LIN {X 0,Y 446.701,Z 503.839,A -85,B 0,C 180,E1 -8817.295,E2 -8817.295} C_VEL
LIN {X 0,Y 446.785,Z 503.811,A -85,B 0,C 180,E1 -8820,E2 -8820} C_VEL
LIN {X 0,Y 446.702,Z 503.837,A -85,B 0,C 180,E1 -8822.706,E2 -8822.706} C_VEL
LIN {X 0,Y 446.643,Z 503.843,A -85,B 0,C 180,E1 -8826.324,E2 -8826.324} C_VEL
LIN {X 0,Y 446.53,Z 503.851,A -85,B 0,C 180,E1 -8829.056,E2 -8829.056} C_VEL
LIN {X 0,Y 446.513,Z 503.865,A -85,B 0,C 180,E1 -8832.73,E2 -8832.73} C_VEL
LIN {X 0,Y 446.488,Z 503.852,A -85,B 0,C 180,E1 -8836.228,E2 -8836.228} C_VEL
LIN {X 0,Y 446.462,Z 503.873,A -85,B 0,C 180,E1 -8839.304,E2 -8839.304} C_VEL
LIN {X 0,Y 446.41,Z 503.87,A -85,B 0,C 180,E1 -8842.2,E2 -8842.2} C_VEL
LIN {X 0,Y 446.452,Z 503.872,A -85,B 0,C 180,E1 -8845.153,E2 -8845.153} C_VEL
LIN {X 0,Y 446.478,Z 503.864,A -85,B 0,C 180,E1 -8848.18,E2 -8848.18} C_VEL
LIN {X 0,Y 446.428,Z 503.877,A -85,B 0,C 180,E1 -8851.3,E2 -8851.3} C_VEL
LIN {X 0,Y 446.426,Z 503.872,A -85,B 0,C 180,E1 -8854.524,E2 -8854.524} C_VEL
LIN {X 0,Y 446.427,Z 503.874,A -85,B 0,C 180,E1 -8858.083,E2 -8858.083} C_VEL
LIN {X 0,Y 446.424,Z 503.878,A -85,B 0,C 180,E1 -8860.919,E2 -8860.919} C_VEL
LIN {X 0,Y 446.421,Z 503.873,A -85,B 0,C 180,E1 -8863.844,E2 -8863.844} C_VEL
LIN {X 0,Y 446.422,Z 503.876,A -85,B 0,C 180,E1 -8866.401,E2 -8866.401} C_VEL
LIN {X 0,Y 446.447,Z 503.87,A -85,B 0,C 180,E1 -8869.804,E2 -8869.804} C_VEL
LIN {X 0,Y 446.409,Z 503.874,A -85,B 0,C 180,E1 -8872.122,E2 -8872.122} C_VEL
LIN {X 0,Y 446.429,Z 503.873,A -85,B 0,C 180,E1 -8875.478,E2 -8875.478} C_VEL
LIN {X 0,Y 446.417,Z 503.875,A -85,B 0,C 180,E1 -8878.701,E2 -8878.701} C_VEL
LIN {X 0,Y 446.486,Z 503.868,A -85,B 0,C 180,E1 -8881.822,E2 -8881.822} C_VEL
LIN {X 0,Y 446.529,Z 503.926,A -85,B 0,C 180,E1 -8882.431,E2 -8882.431} C_VEL
LIN {X 0,Y 448.673,Z 514.714,A -85,B 0,C 180,E1 -8884.485,E2 -8884.485} C_VEL
LIN {X 0,Y 448.915,Z 519.545,A -85,B 0,C 180,E1 -8885.368,E2 -8885.368} C_VEL
LIN {X 0,Y 448.25,Z 538.154,A -85,B 0,C 180,E1 -8888.622,E2 -8888.622} C_VEL
LIN {X 0,Y 447.958,Z 547.38,A -85,B 0,C 180,E1 -8890.172,E2 -8890.172} C_VEL
LIN {X 0,Y 451.104,Z 565.732,A -85,B 0,C 180,E1 -8890.623,E2 -8890.623} C_VEL
LIN {X 0,Y 450.374,Z 639.656,A -85,B 0,C 180,E1 -8891.807,E2 -8891.807} C_VEL
LIN {X 0,Y 449.624,Z 645.502,A -85,B 0,C 180,E1 -8891.871,E2 -8891.871} C_VEL
LIN {X 0,Y 446.643,Z 654.974,A -85,B 0,C 180,E1 -8891.928,E2 -8891.928} C_VEL
LIN {X 0,Y 443.724,Z 664.359,A -85,B 0,C 180,E1 -8892.063,E2 -8892.063} C_VEL
LIN {X 0,Y 443.009,Z 670.054,A -85,B 0,C 180,E1 -8892.237,E2 -8892.237} C_VEL
LIN {X 0,Y 442.573,Z 683.413,A -85,B 0,C 180,E1 -8892.857,E2 -8892.857} C_VEL
LIN {X 0,Y 441.986,Z 695.4,A -85,B 0,C 180,E1 -8893.606,E2 -8893.606} C_VEL
LIN {X 0,Y 441.337,Z 706.738,A -85,B 0,C 180,E1 -8894.53,E2 -8894.53} C_VEL
LIN {X 0,Y 440.642,Z 716.953,A -85,B 0,C 180,E1 -8895.57,E2 -8895.57} C_VEL
LIN {X 0,Y 440.123,Z 725.673,A -85,B 0,C 180,E1 -8896.66,E2 -8896.66} C_VEL
LIN {X 0,Y 439.657,Z 734.405,A -85,B 0,C 180,E1 -8898.006,E2 -8898.006} C_VEL
LIN {X 0,Y 439.126,Z 741.667,A -85,B 0,C 180,E1 -8899.394,E2 -8899.394} C_VEL
LIN {X 0,Y 438.802,Z 747.491,A -85,B 0,C 180,E1 -8900.784,E2 -8900.784} C_VEL
LIN {X 0,Y 438.596,Z 752.07,A -85,B 0,C 180,E1 -8902.172,E2 -8902.172} C_VEL
LIN {X 0,Y 438.466,Z 755.655,A -85,B 0,C 180,E1 -8903.608,E2 -8903.608} C_VEL
LIN {X 0,Y 438.396,Z 757.307,A -85,B 0,C 180,E1 -8904.481,E2 -8904.481} C_VEL
LIN {X 0,Y 438.271,Z 759.557,A -85,B 0,C 180,E1 -8906.322,E2 -8906.322} C_VEL
LIN {X 0,Y 438.355,Z 760.102,A -85,B 0,C 180,E1 -8907.243,E2 -8907.243} C_VEL
LIN {X 0,Y 438.296,Z 760.224,A -85,B 0,C 180,E1 -8908.162,E2 -8908.162} C_VEL
LIN {X 0,Y 438.256,Z 759.301,A -85,B 0,C 180,E1 -8910,E2 -8910} C_VEL
LIN {X 0,Y 438.264,Z 758.263,A -85,B 0,C 180,E1 -8910.919,E2 -8910.919} C_VEL
LIN {X 0,Y 438.373,Z 756.774,A -85,B 0,C 180,E1 -8911.837,E2 -8911.837} C_VEL
LIN {X 0,Y 438.55,Z 753.771,A -85,B 0,C 180,E1 -8913.215,E2 -8913.215} C_VEL
LIN {X 0,Y 438.677,Z 749.73,A -85,B 0,C 180,E1 -8914.594,E2 -8914.594} C_VEL
LIN {X 0,Y 438.925,Z 744.532,A -85,B 0,C 180,E1 -8915.974,E2 -8915.974} C_VEL
LIN {X 0,Y 439.352,Z 738.014,A -85,B 0,C 180,E1 -8917.352,E2 -8917.352} C_VEL
LIN {X 0,Y 439.795,Z 729.922,A -85,B 0,C 180,E1 -8918.732,E2 -8918.732} C_VEL
LIN {X 0,Y 440.32,Z 721.586,A -85,B 0,C 180,E1 -8919.88,E2 -8919.88} C_VEL
LIN {X 0,Y 441.004,Z 711.36,A -85,B 0,C 180,E1 -8921.025,E2 -8921.025} C_VEL
LIN {X 0,Y 441.496,Z 701.275,A -85,B 0,C 180,E1 -8921.943,E2 -8921.943} C_VEL
LIN {X 0,Y 442.074,Z 690.211,A -85,B 0,C 180,E1 -8922.743,E2 -8922.743} C_VEL
LIN {X 0,Y 442.675,Z 677.742,A -85,B 0,C 180,E1 -8923.426,E2 -8923.426} C_VEL
LIN {X 0,Y 443.015,Z 664.927,A -85,B 0,C 180,E1 -8923.935,E2 -8923.935} C_VEL
LIN {X 0,Y 443.262,Z 651.37,A -85,B 0,C 180,E1 -8924.265,E2 -8924.265} C_VEL
LIN {X 0,Y 444.008,Z 565.064,A -85,B 0,C 180,E1 -8925.668,E2 -8925.668} C_VEL
LIN {X 0,Y 440.929,Z 547.62,A -85,B 0,C 180,E1 -8926.085,E2 -8926.085} C_VEL
LIN {X 0,Y 441.452,Z 530.278,A -85,B 0,C 180,E1 -8929.048,E2 -8929.048} C_VEL
LIN {X 0,Y 441.954,Z 517.971,A -85,B 0,C 180,E1 -8931.209,E2 -8931.209} C_VEL
LIN {X 0,Y 439.439,Z 504.755,A -85,B 0,C 180,E1 -8933.719,E2 -8933.719} C_VEL
LIN {X 0,Y 439.431,Z 504.751,A -85,B 0,C 180,E1 -8936.603,E2 -8936.603} C_VEL
LIN {X 0,Y 439.384,Z 504.754,A -85,B 0,C 180,E1 -8939.725,E2 -8939.725} C_VEL
LIN {X 0,Y 439.374,Z 504.757,A -85,B 0,C 180,E1 -8942.945,E2 -8942.945} C_VEL
LIN {X 0,Y 439.373,Z 504.752,A -85,B 0,C 180,E1 -8946.286,E2 -8946.286} C_VEL
LIN {X 0,Y 439.4,Z 504.745,A -85,B 0,C 180,E1 -8949.848,E2 -8949.848} C_VEL
LIN {X 0,Y 439.398,Z 504.753,A -85,B 0,C 180,E1 -8952.628,E2 -8952.628} C_VEL
LIN {X 0,Y 439.405,Z 504.744,A -85,B 0,C 180,E1 -8955.271,E2 -8955.271} C_VEL
LIN {X 0,Y 439.386,Z 504.756,A -85,B 0,C 180,E1 -8958.742,E2 -8958.742} C_VEL
LIN {X 0,Y 439.381,Z 504.752,A -85,B 0,C 180,E1 -8961.605,E2 -8961.605} C_VEL
LIN {X 0,Y 439.396,Z 504.755,A -85,B 0,C 180,E1 -8964.843,E2 -8964.843} C_VEL
LIN {X 0,Y 439.455,Z 504.746,A -85,B 0,C 180,E1 -8966.016,E2 -8966.016} C_VEL
LIN {X 0,Y 443.719,Z 518.661,A -85,B 0,C 180,E1 -8966.455,E2 -8966.455} C_VEL
LIN {X 0,Y 444.068,Z 521.82,A -85,B 0,C 180,E1 -8966.527,E2 -8966.527} C_VEL
LIN {X 0,Y 442.839,Z 611.676,A -85,B 0,C 180,E1 -8968.15,E2 -8968.15} C_VEL
LIN {X 0,Y 442.549,Z 625.742,A -85,B 0,C 180,E1 -8968.604,E2 -8968.604} C_VEL
LIN {X 0,Y 442.193,Z 638.28,A -85,B 0,C 180,E1 -8969.204,E2 -8969.204} C_VEL
LIN {X 0,Y 441.679,Z 649.543,A -85,B 0,C 180,E1 -8969.918,E2 -8969.918} C_VEL
LIN {X 0,Y 441.128,Z 661.441,A -85,B 0,C 180,E1 -8970.883,E2 -8970.883} C_VEL
LIN {X 0,Y 440.621,Z 671.687,A -85,B 0,C 180,E1 -8971.931,E2 -8971.931} C_VEL
LIN {X 0,Y 440.071,Z 681.545,A -85,B 0,C 180,E1 -8973.182,E2 -8973.182} C_VEL
LIN {X 0,Y 439.609,Z 689.541,A -85,B 0,C 180,E1 -8974.427,E2 -8974.427} C_VEL
LIN {X 0,Y 439.275,Z 696.549,A -85,B 0,C 180,E1 -8975.773,E2 -8975.773} C_VEL
LIN {X 0,Y 439.002,Z 701.366,A -85,B 0,C 180,E1 -8976.907,E2 -8976.907} C_VEL
LIN {X 0,Y 438.794,Z 706.406,A -85,B 0,C 180,E1 -8978.384,E2 -8978.384} C_VEL
LIN {X 0,Y 438.609,Z 710.13,A -85,B 0,C 180,E1 -8979.848,E2 -8979.848} C_VEL
LIN {X 0,Y 438.443,Z 712.707,A -85,B 0,C 180,E1 -8981.301,E2 -8981.301} C_VEL
LIN {X 0,Y 438.377,Z 713.822,A -85,B 0,C 180,E1 -8982.265,E2 -8982.265} C_VEL
LIN {X 0,Y 438.384,Z 714.51,A -85,B 0,C 180,E1 -8983.227,E2 -8983.227} C_VEL
LIN {X 0,Y 438.393,Z 714.74,A -85,B 0,C 180,E1 -8984.185,E2 -8984.185} C_VEL
LIN {X 0,Y 438.388,Z 714.513,A -85,B 0,C 180,E1 -8985.137,E2 -8985.137} C_VEL
LIN {X 0,Y 438.443,Z 713.872,A -85,B 0,C 180,E1 -8986.087,E2 -8986.087} C_VEL
LIN {X 0,Y 438.606,Z 711.588,A -85,B 0,C 180,E1 -8987.798,E2 -8987.798} C_VEL
LIN {X 0,Y 438.817,Z 708.09,A -85,B 0,C 180,E1 -8989.386,E2 -8989.386} C_VEL
LIN {X 0,Y 439.028,Z 703.85,A -85,B 0,C 180,E1 -8990.788,E2 -8990.788} C_VEL
LIN {X 0,Y 439.373,Z 698.201,A -85,B 0,C 180,E1 -8992.232,E2 -8992.232} C_VEL
LIN {X 0,Y 439.806,Z 691.572,A -85,B 0,C 180,E1 -8993.577,E2 -8993.577} C_VEL
LIN {X 0,Y 440.275,Z 683.036,A -85,B 0,C 180,E1 -8994.963,E2 -8994.963} C_VEL
LIN {X 0,Y 440.812,Z 674.257,A -85,B 0,C 180,E1 -8996.114,E2 -8996.114} C_VEL
LIN {X 0,Y 441.367,Z 663.485,A -85,B 0,C 180,E1 -8997.262,E2 -8997.262} C_VEL
LIN {X 0,Y 441.962,Z 652.565,A -85,B 0,C 180,E1 -8998.177,E2 -8998.177} C_VEL
LIN {X 0,Y 442.557,Z 640.376,A -85,B 0,C 180,E1 -8998.976,E2 -8998.976} C_VEL
LIN {X 0,Y 442.923,Z 627.861,A -85,B 0,C 180,E1 -8999.592,E2 -8999.592} C_VEL
LIN {X 0,Y 443.21,Z 615.153,A -85,B 0,C 180,E1 -9000.022,E2 -9000.022} C_VEL
LIN {X 0,Y 443.443,Z 594.465,A -85,B 0,C 180,E1 -9000.437,E2 -9000.437} C_VEL
LIN {X 0,Y 444.597,Z 520.546,A -85,B 0,C 180,E1 -9001.826,E2 -9001.826} C_VEL
LIN {X 0,Y 443.026,Z 515.39,A -85,B 0,C 180,E1 -9002.01,E2 -9002.01} C_VEL
LIN {X 0,Y 440.276,Z 508.037,A -85,B 0,C 180,E1 -9002.302,E2 -9002.302} C_VEL
LIN {X 0,Y 439.499,Z 504.741,A -85,B 0,C 180,E1 -9003.323,E2 -9003.323} C_VEL
LIN {X 0,Y 439.614,Z 504.725,A -85,B 0,C 180,E1 -9006.425,E2 -9006.425} C_VEL
LIN {X 0,Y 439.493,Z 504.743,A -85,B 0,C 180,E1 -9009.202,E2 -9009.202} C_VEL
LIN {X 0,Y 439.495,Z 504.739,A -85,B 0,C 180,E1 -9012.727,E2 -9012.727} C_VEL
LIN {X 0,Y 439.438,Z 504.745,A -85,B 0,C 180,E1 -9016.349,E2 -9016.349} C_VEL
LIN {X 0,Y 439.394,Z 504.751,A -85,B 0,C 180,E1 -9019.627,E2 -9019.627} C_VEL
LIN {X 0,Y 439.357,Z 504.756,A -85,B 0,C 180,E1 -9022.576,E2 -9022.576} C_VEL
LIN {X 0,Y 439.397,Z 504.749,A -85,B 0,C 180,E1 -9025.585,E2 -9025.585} C_VEL
LIN {X 0,Y 439.418,Z 504.746,A -85,B 0,C 180,E1 -9028.673,E2 -9028.673} C_VEL
LIN {X 0,Y 439.367,Z 504.75,A -85,B 0,C 180,E1 -9031.861,E2 -9031.861} C_VEL
LIN {X 0,Y 439.394,Z 504.753,A -85,B 0,C 180,E1 -9035.156,E2 -9035.156} C_VEL
LIN {X 0,Y 439.384,Z 504.751,A -85,B 0,C 180,E1 -9038.595,E2 -9038.595} C_VEL
LIN {X 0,Y 439.383,Z 504.755,A -85,B 0,C 180,E1 -9041.257,E2 -9041.257} C_VEL
LIN {X 0,Y 439.397,Z 504.753,A -85,B 0,C 180,E1 -9044.73,E2 -9044.73} C_VEL
LIN {X 0,Y 439.394,Z 504.752,A -85,B 0,C 180,E1 -9047.797,E2 -9047.797} C_VEL
LIN {X 0,Y 439.427,Z 504.749,A -85,B 0,C 180,E1 -9050.229,E2 -9050.229} C_VEL
LIN {X 0,Y 439.374,Z 504.754,A -85,B 0,C 180,E1 -9053.714,E2 -9053.714} C_VEL
LIN {X 0,Y 439.371,Z 504.761,A -85,B 0,C 180,E1 -9057.055,E2 -9057.055} C_VEL
LIN {X 0,Y 439.434,Z 504.811,A -85,B 0,C 180,E1 -9060.887,E2 -9060.887} C_VEL
LIN {X 0,Y 441.948,Z 516.24,A -85,B 0,C 180,E1 -9063.169,E2 -9063.169} C_VEL
LIN {X 0,Y 442.844,Z 522.646,A -85,B 0,C 180,E1 -9064.377,E2 -9064.377} C_VEL
LIN {X 0,Y 441.66,Z 542.589,A -85,B 0,C 180,E1 -9067.795,E2 -9067.795} C_VEL
LIN {X 0,Y 440.607,Z 562.702,A -85,B 0,C 180,E1 -9071.156,E2 -9071.156} C_VEL
LIN {X 0,Y 440.45,Z 566.137,A -85,B 0,C 180,E1 -9071.705,E2 -9071.705} C_VEL
LIN {X 0,Y 443.689,Z 590.86,A -85,B 0,C 180,E1 -9072.348,E2 -9072.348} C_VEL
LIN {X 0,Y 443.939,Z 596.387,A -85,B 0,C 180,E1 -9072.466,E2 -9072.466} C_VEL
LIN {X 0,Y 442.814,Z 677.088,A -85,B 0,C 180,E1 -9073.963,E2 -9073.963} C_VEL
LIN {X 0,Y 442.19,Z 695.595,A -85,B 0,C 180,E1 -9074.561,E2 -9074.561} C_VEL
LIN {X 0,Y 441.694,Z 707.963,A -85,B 0,C 180,E1 -9075.134,E2 -9075.134} C_VEL
LIN {X 0,Y 441.141,Z 718.982,A -85,B 0,C 180,E1 -9075.822,E2 -9075.822} C_VEL
LIN {X 0,Y 440.644,Z 730.447,A -85,B 0,C 180,E1 -9076.745,E2 -9076.745} C_VEL
LIN {X 0,Y 440.053,Z 740.763,A -85,B 0,C 180,E1 -9077.783,E2 -9077.783} C_VEL
LIN {X 0,Y 439.487,Z 749.99,A -85,B 0,C 180,E1 -9078.937,E2 -9078.937} C_VEL
LIN {X 0,Y 439.03,Z 758.938,A -85,B 0,C 180,E1 -9080.324,E2 -9080.324} C_VEL
LIN {X 0,Y 438.735,Z 766.108,A -85,B 0,C 180,E1 -9081.711,E2 -9081.711} C_VEL
LIN {X 0,Y 438.52,Z 771.792,A -85,B 0,C 180,E1 -9083.097,E2 -9083.097} C_VEL
LIN {X 0,Y 438.431,Z 776.248,A -85,B 0,C 180,E1 -9084.481,E2 -9084.481} C_VEL
LIN {X 0,Y 438.378,Z 778.591,A -85,B 0,C 180,E1 -9085.402,E2 -9085.402} C_VEL
LIN {X 0,Y 438.308,Z 780.499,A -85,B 0,C 180,E1 -9086.323,E2 -9086.323} C_VEL
LIN {X 0,Y 438.417,Z 781.956,A -85,B 0,C 180,E1 -9087.244,E2 -9087.244} C_VEL
LIN {X 0,Y 438.263,Z 783.597,A -85,B 0,C 180,E1 -9089.081,E2 -9089.081} C_VEL
LIN {X 0,Y 438.266,Z 783.831,A -85,B 0,C 180,E1 -9090,E2 -9090} C_VEL
LIN {X 0,Y 438.262,Z 783.624,A -85,B 0,C 180,E1 -9090.919,E2 -9090.919} C_VEL
LIN {X 0,Y 438.419,Z 782.018,A -85,B 0,C 180,E1 -9092.756,E2 -9092.756} C_VEL
LIN {X 0,Y 438.312,Z 780.602,A -85,B 0,C 180,E1 -9093.677,E2 -9093.677} C_VEL
LIN {X 0,Y 438.432,Z 777.642,A -85,B 0,C 180,E1 -9095.058,E2 -9095.058} C_VEL
LIN {X 0,Y 438.471,Z 773.619,A -85,B 0,C 180,E1 -9096.442,E2 -9096.442} C_VEL
LIN {X 0,Y 438.686,Z 767.398,A -85,B 0,C 180,E1 -9098.058,E2 -9098.058} C_VEL
LIN {X 0,Y 439.013,Z 760.611,A -85,B 0,C 180,E1 -9099.444,E2 -9099.444} C_VEL
LIN {X 0,Y 439.431,Z 752.134,A -85,B 0,C 180,E1 -9100.831,E2 -9100.831} C_VEL
LIN {X 0,Y 439.956,Z 743.389,A -85,B 0,C 180,E1 -9101.985,E2 -9101.985} C_VEL
LIN {X 0,Y 440.532,Z 733.532,A -85,B 0,C 180,E1 -9103.047,E2 -9103.047} C_VEL
LIN {X 0,Y 441.063,Z 723.244,A -85,B 0,C 180,E1 -9103.946,E2 -9103.946} C_VEL
LIN {X 0,Y 441.657,Z 711.46,A -85,B 0,C 180,E1 -9104.75,E2 -9104.75} C_VEL
LIN {X 0,Y 442.178,Z 699.172,A -85,B 0,C 180,E1 -9105.38,E2 -9105.38} C_VEL
LIN {X 0,Y 442.641,Z 686.478,A -85,B 0,C 180,E1 -9105.836,E2 -9105.836} C_VEL
LIN {X 0,Y 442.895,Z 672.991,A -85,B 0,C 180,E1 -9106.122,E2 -9106.122} C_VEL
LIN {X 0,Y 443.536,Z 608.774,A -85,B 0,C 180,E1 -9107.2,E2 -9107.2} C_VEL
LIN {X 0,Y 443.59,Z 591.986,A -85,B 0,C 180,E1 -9107.509,E2 -9107.509} C_VEL
LIN {X 0,Y 440.47,Z 568.609,A -85,B 0,C 180,E1 -9108.079,E2 -9108.079} C_VEL
LIN {X 0,Y 441.403,Z 549.446,A -85,B 0,C 180,E1 -9111.236,E2 -9111.236} C_VEL
LIN {X 0,Y 442.511,Z 530.547,A -85,B 0,C 180,E1 -9114.389,E2 -9114.389} C_VEL
LIN {X 0,Y 442.898,Z 521.782,A -85,B 0,C 180,E1 -9115.872,E2 -9115.872} C_VEL
LIN {X 0,Y 440.519,Z 509.778,A -85,B 0,C 180,E1 -9118.075,E2 -9118.075} C_VEL
LIN {X 0,Y 439.443,Z 504.749,A -85,B 0,C 180,E1 -9119.063,E2 -9119.063} C_VEL
LIN {X 0,Y 439.371,Z 504.758,A -85,B 0,C 180,E1 -9122.945,E2 -9122.945} C_VEL
LIN {X 0,Y 439.371,Z 504.749,A -85,B 0,C 180,E1 -9126.286,E2 -9126.286} C_VEL
LIN {X 0,Y 439.41,Z 504.745,A -85,B 0,C 180,E1 -9129.85,E2 -9129.85} C_VEL
LIN {X 0,Y 439.383,Z 504.753,A -85,B 0,C 180,E1 -9132.627,E2 -9132.627} C_VEL
LIN {X 0,Y 439.398,Z 504.755,A -85,B 0,C 180,E1 -9135.27,E2 -9135.27} C_VEL
LIN {X 0,Y 439.393,Z 504.745,A -85,B 0,C 180,E1 -9138.741,E2 -9138.741} C_VEL
LIN {X 0,Y 439.385,Z 504.75,A -85,B 0,C 180,E1 -9141.604,E2 -9141.604} C_VEL
LIN {X 0,Y 439.394,Z 504.747,A -85,B 0,C 180,E1 -9144.844,E2 -9144.844} C_VEL
LIN {X 0,Y 439.367,Z 504.747,A -85,B 0,C 180,E1 -9148.139,E2 -9148.139} C_VEL
LIN {X 0,Y 439.418,Z 504.751,A -85,B 0,C 180,E1 -9151.327,E2 -9151.327} C_VEL
LIN {X 0,Y 439.397,Z 504.745,A -85,B 0,C 180,E1 -9154.415,E2 -9154.415} C_VEL
LIN {X 0,Y 439.356,Z 504.753,A -85,B 0,C 180,E1 -9157.424,E2 -9157.424} C_VEL
LIN {X 0,Y 439.433,Z 504.745,A -85,B 0,C 180,E1 -9160.662,E2 -9160.662} C_VEL
LIN {X 0,Y 439.453,Z 504.73,A -85,B 0,C 180,E1 -9164.224,E2 -9164.224} C_VEL
LIN {X 0,Y 439.499,Z 504.735,A -85,B 0,C 180,E1 -9168.002,E2 -9168.002} C_VEL
LIN {X 0,Y 439.539,Z 504.718,A -85,B 0,C 180,E1 -9171.726,E2 -9171.726} C_VEL
LIN {X 0,Y 439.619,Z 504.719,A -85,B 0,C 180,E1 -9174.496,E2 -9174.496} C_VEL
LIN {X 0,Y 439.627,Z 504.715,A -85,B 0,C 180,E1 -9178.168,E2 -9178.168} C_VEL
LIN {X 0,Y 439.755,Z 504.686,A -85,B 0,C 180,E1 -9180,E2 -9180} C_VEL
LIN {X 0,Y 439.649,Z 504.716,A -85,B 0,C 180,E1 -9182.749,E2 -9182.749} C_VEL
LIN {X 0,Y 439.614,Z 504.719,A -85,B 0,C 180,E1 -9186.426,E2 -9186.426} C_VEL
LIN {X 0,Y 439.492,Z 504.729,A -85,B 0,C 180,E1 -9189.202,E2 -9189.202} C_VEL
LIN {X 0,Y 439.457,Z 504.747,A -85,B 0,C 180,E1 -9192.938,E2 -9192.938} C_VEL
LIN {X 0,Y 439.439,Z 504.73,A -85,B 0,C 180,E1 -9196.349,E2 -9196.349} C_VEL
LIN {X 0,Y 439.395,Z 504.75,A -85,B 0,C 180,E1 -9199.627,E2 -9199.627} C_VEL
LIN {X 0,Y 439.357,Z 504.751,A -85,B 0,C 180,E1 -9202.576,E2 -9202.576} C_VEL
LIN {X 0,Y 439.399,Z 504.75,A -85,B 0,C 180,E1 -9205.586,E2 -9205.586} C_VEL
LIN {X 0,Y 439.419,Z 504.746,A -85,B 0,C 180,E1 -9208.674,E2 -9208.674} C_VEL
LIN {X 0,Y 439.379,Z 504.751,A -85,B 0,C 180,E1 -9212.034,E2 -9212.034} C_VEL
LIN {X 0,Y 439.392,Z 504.75,A -85,B 0,C 180,E1 -9215.342,E2 -9215.342} C_VEL
LIN {X 0,Y 439.385,Z 504.754,A -85,B 0,C 180,E1 -9218.595,E2 -9218.595} C_VEL
LIN {X 0,Y 439.385,Z 504.758,A -85,B 0,C 180,E1 -9221.258,E2 -9221.258} C_VEL
LIN {X 0,Y 439.404,Z 504.751,A -85,B 0,C 180,E1 -9224.729,E2 -9224.729} C_VEL
LIN {X 0,Y 439.397,Z 504.749,A -85,B 0,C 180,E1 -9227.797,E2 -9227.797} C_VEL
LIN {X 0,Y 439.429,Z 504.744,A -85,B 0,C 180,E1 -9230.229,E2 -9230.229} C_VEL
LIN {X 0,Y 439.373,Z 504.752,A -85,B 0,C 180,E1 -9233.714,E2 -9233.714} C_VEL
LIN {X 0,Y 439.373,Z 504.755,A -85,B 0,C 180,E1 -9237.055,E2 -9237.055} C_VEL
LIN {X 0,Y 439.384,Z 504.752,A -85,B 0,C 180,E1 -9240.275,E2 -9240.275} C_VEL
LIN {X 0,Y 439.482,Z 504.873,A -85,B 0,C 180,E1 -9242.194,E2 -9242.194} C_VEL
LIN {X 0,Y 441.934,Z 517.239,A -85,B 0,C 180,E1 -9244.573,E2 -9244.573} C_VEL
LIN {X 0,Y 441.822,Z 525.514,A -85,B 0,C 180,E1 -9246.07,E2 -9246.07} C_VEL
LIN {X 0,Y 441.178,Z 542.313,A -85,B 0,C 180,E1 -9248.997,E2 -9248.997} C_VEL
LIN {X 0,Y 441.052,Z 547.544,A -85,B 0,C 180,E1 -9249.879,E2 -9249.879} C_VEL
LIN {X 0,Y 444.354,Z 565.884,A -85,B 0,C 180,E1 -9250.34,E2 -9250.34} C_VEL
LIN {X 0,Y 443.385,Z 656.466,A -85,B 0,C 180,E1 -9251.834,E2 -9251.834} C_VEL
LIN {X 0,Y 443.021,Z 669.411,A -85,B 0,C 180,E1 -9252.214,E2 -9252.214} C_VEL
LIN {X 0,Y 443.009,Z 670.054,A -85,B 0,C 180,E1 -9252.237,E2 -9252.237} C_VEL
LIN {X 0,Y 442.219,Z 675.707,A -85,B 0,C 180,E1 -9252.44,E2 -9252.44} C_VEL
LIN {X 0,Y 439.059,Z 684.741,A -85,B 0,C 180,E1 -9252.79,E2 -9252.79} C_VEL
LIN {X 0,Y 435.844,Z 693.491,A -85,B 0,C 180,E1 -9253.239,E2 -9253.239} C_VEL
LIN {X 0,Y 434.972,Z 698.627,A -85,B 0,C 180,E1 -9253.597,E2 -9253.597} C_VEL
LIN {X 0,Y 434.304,Z 709.182,A -85,B 0,C 180,E1 -9254.514,E2 -9254.514} C_VEL
LIN {X 0,Y 433.676,Z 717.981,A -85,B 0,C 180,E1 -9255.453,E2 -9255.453} C_VEL
LIN {X 0,Y 433.108,Z 727.033,A -85,B 0,C 180,E1 -9256.631,E2 -9256.631} C_VEL
LIN {X 0,Y 432.578,Z 735.79,A -85,B 0,C 180,E1 -9258.045,E2 -9258.045} C_VEL
LIN {X 0,Y 432.029,Z 742.845,A -85,B 0,C 180,E1 -9259.455,E2 -9259.455} C_VEL
LIN {X 0,Y 431.749,Z 747.598,A -85,B 0,C 180,E1 -9260.632,E2 -9260.632} C_VEL
LIN {X 0,Y 431.525,Z 752.195,A -85,B 0,C 180,E1 -9262.043,E2 -9262.043} C_VEL
LIN {X 0,Y 431.373,Z 756.075,A -85,B 0,C 180,E1 -9263.633,E2 -9263.633} C_VEL
LIN {X 0,Y 431.234,Z 758.791,A -85,B 0,C 180,E1 -9265.326,E2 -9265.326} C_VEL
LIN {X 0,Y 431.263,Z 760.283,A -85,B 0,C 180,E1 -9267.198,E2 -9267.198} C_VEL
LIN {X 0,Y 431.22,Z 760.418,A -85,B 0,C 180,E1 -9268.132,E2 -9268.132} C_VEL
LIN {X 0,Y 431.17,Z 759.51,A -85,B 0,C 180,E1 -9270,E2 -9270} C_VEL
LIN {X 0,Y 431.182,Z 758.482,A -85,B 0,C 180,E1 -9270.934,E2 -9270.934} C_VEL
LIN {X 0,Y 431.294,Z 757.005,A -85,B 0,C 180,E1 -9271.868,E2 -9271.868} C_VEL
LIN {X 0,Y 431.483,Z 754.016,A -85,B 0,C 180,E1 -9273.268,E2 -9273.268} C_VEL
LIN {X 0,Y 431.598,Z 749.992,A -85,B 0,C 180,E1 -9274.67,E2 -9274.67} C_VEL
LIN {X 0,Y 431.884,Z 744.811,A -85,B 0,C 180,E1 -9276.072,E2 -9276.072} C_VEL
LIN {X 0,Y 432.32,Z 738.311,A -85,B 0,C 180,E1 -9277.472,E2 -9277.472} C_VEL
LIN {X 0,Y 432.794,Z 730.246,A -85,B 0,C 180,E1 -9278.874,E2 -9278.874} C_VEL
LIN {X 0,Y 433.351,Z 721.941,A -85,B 0,C 180,E1 -9280.04,E2 -9280.04} C_VEL
LIN {X 0,Y 434.053,Z 711.745,A -85,B 0,C 180,E1 -9281.203,E2 -9281.203} C_VEL
LIN {X 0,Y 434.565,Z 701.699,A -85,B 0,C 180,E1 -9282.136,E2 -9282.136} C_VEL
LIN {X 0,Y 435.186,Z 690.712,A -85,B 0,C 180,E1 -9282.948,E2 -9282.948} C_VEL
LIN {X 0,Y 435.798,Z 678.336,A -85,B 0,C 180,E1 -9283.642,E2 -9283.642} C_VEL
LIN {X 0,Y 436.183,Z 665.11,A -85,B 0,C 180,E1 -9284.177,E2 -9284.177} C_VEL
LIN {X 0,Y 436.411,Z 652.341,A -85,B 0,C 180,E1 -9284.498,E2 -9284.498} C_VEL
LIN {X 0,Y 437.299,Z 566.356,A -85,B 0,C 180,E1 -9285.915,E2 -9285.915} C_VEL
LIN {X 0,Y 434.044,Z 547.715,A -85,B 0,C 180,E1 -9286.37,E2 -9286.37} C_VEL
LIN {X 0,Y 434.548,Z 530.393,A -85,B 0,C 180,E1 -9289.362,E2 -9289.362} C_VEL
LIN {X 0,Y 435.03,Z 519.325,A -85,B 0,C 180,E1 -9291.314,E2 -9291.314} C_VEL
LIN {X 0,Y 432.4,Z 505.631,A -85,B 0,C 180,E1 -9293.974,E2 -9293.974} C_VEL
LIN {X 0,Y 432.393,Z 505.626,A -85,B 0,C 180,E1 -9297.071,E2 -9297.071} C_VEL
LIN {X 0,Y 432.349,Z 505.632,A -85,B 0,C 180,E1 -9300.51,E2 -9300.51} C_VEL
LIN {X 0,Y 432.36,Z 505.624,A -85,B 0,C 180,E1 -9304.003,E2 -9304.003} C_VEL
LIN {X 0,Y 432.322,Z 505.633,A -85,B 0,C 180,E1 -9307.196,E2 -9307.196} C_VEL
LIN {X 0,Y 432.332,Z 505.626,A -85,B 0,C 180,E1 -9310.178,E2 -9310.178} C_VEL
LIN {X 0,Y 432.362,Z 505.629,A -85,B 0,C 180,E1 -9313.054,E2 -9313.054} C_VEL
LIN {X 0,Y 432.34,Z 505.622,A -85,B 0,C 180,E1 -9315.662,E2 -9315.662} C_VEL
LIN {X 0,Y 432.331,Z 505.632,A -85,B 0,C 180,E1 -9318.397,E2 -9318.397} C_VEL
LIN {X 0,Y 432.343,Z 505.628,A -85,B 0,C 180,E1 -9321.85,E2 -9321.85} C_VEL
LIN {X 0,Y 432.352,Z 505.631,A -85,B 0,C 180,E1 -9325.324,E2 -9325.324} C_VEL
LIN {X 0,Y 432.38,Z 505.626,A -85,B 0,C 180,E1 -9325.747,E2 -9325.747} C_VEL
LIN {X 0,Y 436.927,Z 519.644,A -85,B 0,C 180,E1 -9326.21,E2 -9326.21} C_VEL
LIN {X 0,Y 437.213,Z 524.529,A -85,B 0,C 180,E1 -9326.314,E2 -9326.314} C_VEL
LIN {X 0,Y 435.961,Z 612.071,A -85,B 0,C 180,E1 -9327.928,E2 -9327.928} C_VEL
LIN {X 0,Y 435.658,Z 625.901,A -85,B 0,C 180,E1 -9328.38,E2 -9328.38} C_VEL
LIN {X 0,Y 435.28,Z 639.165,A -85,B 0,C 180,E1 -9329.025,E2 -9329.025} C_VEL
LIN {X 0,Y 434.729,Z 650.87,A -85,B 0,C 180,E1 -9329.789,E2 -9329.789} C_VEL
LIN {X 0,Y 434.207,Z 661.679,A -85,B 0,C 180,E1 -9330.684,E2 -9330.684} C_VEL
LIN {X 0,Y 433.683,Z 671.641,A -85,B 0,C 180,E1 -9331.705,E2 -9331.705} C_VEL
LIN {X 0,Y 433.114,Z 681.615,A -85,B 0,C 180,E1 -9332.977,E2 -9332.977} C_VEL
LIN {X 0,Y 432.638,Z 689.7,A -85,B 0,C 180,E1 -9334.244,E2 -9334.244} C_VEL
LIN {X 0,Y 432.281,Z 696.569,A -85,B 0,C 180,E1 -9335.564,E2 -9335.564} C_VEL
LIN {X 0,Y 431.928,Z 702.625,A -85,B 0,C 180,E1 -9337.013,E2 -9337.013} C_VEL
LIN {X 0,Y 431.713,Z 707.564,A -85,B 0,C 180,E1 -9338.548,E2 -9338.548} C_VEL
LIN {X 0,Y 431.502,Z 711.051,A -85,B 0,C 180,E1 -9339.999,E2 -9339.999} C_VEL
LIN {X 0,Y 431.412,Z 712.81,A -85,B 0,C 180,E1 -9340.985,E2 -9340.985} C_VEL
LIN {X 0,Y 431.315,Z 714.096,A -85,B 0,C 180,E1 -9341.965,E2 -9341.965} C_VEL
LIN {X 0,Y 431.313,Z 714.89,A -85,B 0,C 180,E1 -9342.944,E2 -9342.944} C_VEL
LIN {X 0,Y 431.338,Z 715.282,A -85,B 0,C 180,E1 -9344.006,E2 -9344.006} C_VEL
LIN {X 0,Y 431.319,Z 715.201,A -85,B 0,C 180,E1 -9344.888,E2 -9344.888} C_VEL
LIN {X 0,Y 431.358,Z 714.664,A -85,B 0,C 180,E1 -9345.854,E2 -9345.854} C_VEL
LIN {X 0,Y 431.44,Z 713.713,A -85,B 0,C 180,E1 -9346.817,E2 -9346.817} C_VEL
LIN {X 0,Y 431.541,Z 712.342,A -85,B 0,C 180,E1 -9347.777,E2 -9347.777} C_VEL
LIN {X 0,Y 431.739,Z 709.401,A -85,B 0,C 180,E1 -9349.21,E2 -9349.21} C_VEL
LIN {X 0,Y 431.976,Z 705.382,A -85,B 0,C 180,E1 -9350.636,E2 -9350.636} C_VEL
LIN {X 0,Y 432.331,Z 699.963,A -85,B 0,C 180,E1 -9352.104,E2 -9352.104} C_VEL
LIN {X 0,Y 432.825,Z 692.367,A -85,B 0,C 180,E1 -9353.707,E2 -9353.707} C_VEL
LIN {X 0,Y 433.255,Z 685.433,A -85,B 0,C 180,E1 -9354.881,E2 -9354.881} C_VEL
LIN {X 0,Y 433.743,Z 677.083,A -85,B 0,C 180,E1 -9356.051,E2 -9356.051} C_VEL
LIN {X 0,Y 434.342,Z 666.757,A -85,B 0,C 180,E1 -9357.217,E2 -9357.217} C_VEL
LIN {X 0,Y 435.039,Z 655.133,A -85,B 0,C 180,E1 -9358.264,E2 -9358.264} C_VEL
LIN {X 0,Y 435.64,Z 643.532,A -85,B 0,C 180,E1 -9359.075,E2 -9359.075} C_VEL
LIN {X 0,Y 436.067,Z 630.242,A -85,B 0,C 180,E1 -9359.781,E2 -9359.781} C_VEL
LIN {X 0,Y 436.387,Z 617.946,A -85,B 0,C 180,E1 -9360.236,E2 -9360.236} C_VEL
LIN {X 0,Y 436.636,Z 601.939,A -85,B 0,C 180,E1 -9360.593,E2 -9360.593} C_VEL
LIN {X 0,Y 437.959,Z 521.791,A -85,B 0,C 180,E1 -9362.134,E2 -9362.134} C_VEL
LIN {X 0,Y 433.961,Z 510.765,A -85,B 0,C 180,E1 -9362.576,E2 -9362.576} C_VEL
LIN {X 0,Y 433.214,Z 508.698,A -85,B 0,C 180,E1 -9362.685,E2 -9362.685} C_VEL
LIN {X 0,Y 432.417,Z 505.623,A -85,B 0,C 180,E1 -9363.611,E2 -9363.611} C_VEL
LIN {X 0,Y 432.567,Z 505.603,A -85,B 0,C 180,E1 -9366.53,E2 -9366.53} C_VEL
LIN {X 0,Y 432.436,Z 505.623,A -85,B 0,C 180,E1 -9369.353,E2 -9369.353} C_VEL
LIN {X 0,Y 432.436,Z 505.619,A -85,B 0,C 180,E1 -9372.812,E2 -9372.812} C_VEL
LIN {X 0,Y 432.403,Z 505.622,A -85,B 0,C 180,E1 -9376.479,E2 -9376.479} C_VEL
LIN {X 0,Y 432.33,Z 505.63,A -85,B 0,C 180,E1 -9379.961,E2 -9379.961} C_VEL
LIN {X 0,Y 432.311,Z 505.637,A -85,B 0,C 180,E1 -9382.965,E2 -9382.965} C_VEL
LIN {X 0,Y 432.357,Z 505.624,A -85,B 0,C 180,E1 -9386.033,E2 -9386.033} C_VEL
LIN {X 0,Y 432.345,Z 505.628,A -85,B 0,C 180,E1 -9389.187,E2 -9389.187} C_VEL
LIN {X 0,Y 432.319,Z 505.628,A -85,B 0,C 180,E1 -9392.294,E2 -9392.294} C_VEL
LIN {X 0,Y 432.334,Z 505.629,A -85,B 0,C 180,E1 -9394.678,E2 -9394.678} C_VEL
LIN {X 0,Y 432.342,Z 505.626,A -85,B 0,C 180,E1 -9398.149,E2 -9398.149} C_VEL
LIN {X 0,Y 432.327,Z 505.63,A -85,B 0,C 180,E1 -9401.603,E2 -9401.603} C_VEL
LIN {X 0,Y 432.329,Z 505.63,A -85,B 0,C 180,E1 -9404.348,E2 -9404.348} C_VEL
LIN {X 0,Y 432.321,Z 505.636,A -85,B 0,C 180,E1 -9407.016,E2 -9407.016} C_VEL
LIN {X 0,Y 432.333,Z 505.632,A -85,B 0,C 180,E1 -9409.821,E2 -9409.821} C_VEL
LIN {X 0,Y 432.313,Z 505.637,A -85,B 0,C 180,E1 -9413.024,E2 -9413.024} C_VEL
LIN {X 0,Y 432.357,Z 505.63,A -85,B 0,C 180,E1 -9415.997,E2 -9415.997} C_VEL
LIN {X 0,Y 432.346,Z 505.636,A -85,B 0,C 180,E1 -9419.49,E2 -9419.49} C_VEL
LIN {X 0,Y 432.396,Z 505.749,A -85,B 0,C 180,E1 -9420.55,E2 -9420.55} C_VEL
LIN {X 0,Y 435.162,Z 518.255,A -85,B 0,C 180,E1 -9423.115,E2 -9423.115} C_VEL
LIN {X 0,Y 435.979,Z 523.907,A -85,B 0,C 180,E1 -9424.2,E2 -9424.2} C_VEL
LIN {X 0,Y 434.728,Z 543.733,A -85,B 0,C 180,E1 -9427.672,E2 -9427.672} C_VEL
LIN {X 0,Y 433.587,Z 563.756,A -85,B 0,C 180,E1 -9431.085,E2 -9431.085} C_VEL
LIN {X 0,Y 433.502,Z 565.361,A -85,B 0,C 180,E1 -9431.351,E2 -9431.351} C_VEL
LIN {X 0,Y 436.318,Z 585.941,A -85,B 0,C 180,E1 -9431.907,E2 -9431.907} C_VEL
LIN {X 0,Y 437.268,Z 594.898,A -85,B 0,C 180,E1 -9432.135,E2 -9432.135} C_VEL
LIN {X 0,Y 436.01,Z 676.887,A -85,B 0,C 180,E1 -9433.706,E2 -9433.706} C_VEL
LIN {X 0,Y 435.348,Z 695.169,A -85,B 0,C 180,E1 -9434.312,E2 -9434.312} C_VEL
LIN {X 0,Y 434.828,Z 707.606,A -85,B 0,C 180,E1 -9434.893,E2 -9434.893} C_VEL
LIN {X 0,Y 434.247,Z 718.665,A -85,B 0,C 180,E1 -9435.592,E2 -9435.592} C_VEL
LIN {X 0,Y 433.69,Z 729.677,A -85,B 0,C 180,E1 -9436.485,E2 -9436.485} C_VEL
LIN {X 0,Y 433.089,Z 740.487,A -85,B 0,C 180,E1 -9437.584,E2 -9437.584} C_VEL
LIN {X 0,Y 432.501,Z 749.733,A -85,B 0,C 180,E1 -9438.756,E2 -9438.756} C_VEL
LIN {X 0,Y 432.005,Z 758.691,A -85,B 0,C 180,E1 -9440.165,E2 -9440.165} C_VEL
LIN {X 0,Y 431.674,Z 765.873,A -85,B 0,C 180,E1 -9441.574,E2 -9441.574} C_VEL
LIN {X 0,Y 431.435,Z 771.568,A -85,B 0,C 180,E1 -9442.983,E2 -9442.983} C_VEL
LIN {X 0,Y 431.334,Z 776.031,A -85,B 0,C 180,E1 -9444.39,E2 -9444.39} C_VEL
LIN {X 0,Y 431.308,Z 778.378,A -85,B 0,C 180,E1 -9445.327,E2 -9445.327} C_VEL
LIN {X 0,Y 431.214,Z 780.289,A -85,B 0,C 180,E1 -9446.262,E2 -9446.262} C_VEL
LIN {X 0,Y 431.321,Z 781.753,A -85,B 0,C 180,E1 -9447.198,E2 -9447.198} C_VEL
LIN {X 0,Y 431.251,Z 782.774,A -85,B 0,C 180,E1 -9448.132,E2 -9448.132} C_VEL
LIN {X 0,Y 431.179,Z 783.64,A -85,B 0,C 180,E1 -9450,E2 -9450} C_VEL
LIN {X 0,Y 431.179,Z 783.439,A -85,B 0,C 180,E1 -9450.934,E2 -9450.934} C_VEL
LIN {X 0,Y 431.251,Z 782.835,A -85,B 0,C 180,E1 -9451.868,E2 -9451.868} C_VEL
LIN {X 0,Y 431.323,Z 781.84,A -85,B 0,C 180,E1 -9452.802,E2 -9452.802} C_VEL
LIN {X 0,Y 431.218,Z 780.429,A -85,B 0,C 180,E1 -9453.738,E2 -9453.738} C_VEL
LIN {X 0,Y 431.345,Z 777.476,A -85,B 0,C 180,E1 -9455.141,E2 -9455.141} C_VEL
LIN {X 0,Y 431.385,Z 773.462,A -85,B 0,C 180,E1 -9456.548,E2 -9456.548} C_VEL
LIN {X 0,Y 431.624,Z 767.253,A -85,B 0,C 180,E1 -9458.191,E2 -9458.191} C_VEL
LIN {X 0,Y 431.971,Z 760.478,A -85,B 0,C 180,E1 -9459.599,E2 -9459.599} C_VEL
LIN {X 0,Y 432.328,Z 753.559,A -85,B 0,C 180,E1 -9460.774,E2 -9460.774} C_VEL
LIN {X 0,Y 432.885,Z 745.211,A -85,B 0,C 180,E1 -9461.946,E2 -9461.946} C_VEL
LIN {X 0,Y 433.499,Z 734.873,A -85,B 0,C 180,E1 -9463.119,E2 -9463.119} C_VEL
LIN {X 0,Y 434.091,Z 724.62,A -85,B 0,C 180,E1 -9464.055,E2 -9464.055} C_VEL
LIN {X 0,Y 434.711,Z 713.374,A -85,B 0,C 180,E1 -9464.871,E2 -9464.871} C_VEL
LIN {X 0,Y 435.228,Z 701.836,A -85,B 0,C 180,E1 -9465.512,E2 -9465.512} C_VEL
LIN {X 0,Y 435.767,Z 688.53,A -85,B 0,C 180,E1 -9466.033,E2 -9466.033} C_VEL
LIN {X 0,Y 436.094,Z 675.356,A -85,B 0,C 180,E1 -9466.351,E2 -9466.351} C_VEL
LIN {X 0,Y 436.871,Z 593.672,A -85,B 0,C 180,E1 -9467.717,E2 -9467.717} C_VEL
LIN {X 0,Y 433.489,Z 568.289,A -85,B 0,C 180,E1 -9468.331,E2 -9468.331} C_VEL
LIN {X 0,Y 434.592,Z 547.402,A -85,B 0,C 180,E1 -9471.835,E2 -9471.835} C_VEL
LIN {X 0,Y 435.76,Z 527.996,A -85,B 0,C 180,E1 -9475.127,E2 -9475.127} C_VEL
LIN {X 0,Y 435.893,Z 522.6,A -85,B 0,C 180,E1 -9476.062,E2 -9476.062} C_VEL
LIN {X 0,Y 433.392,Z 510.177,A -85,B 0,C 180,E1 -9478.392,E2 -9478.392} C_VEL
LIN {X 0,Y 432.384,Z 505.628,A -85,B 0,C 180,E1 -9479.284,E2 -9479.284} C_VEL
LIN {X 0,Y 432.321,Z 505.633,A -85,B 0,C 180,E1 -9482.442,E2 -9482.442} C_VEL
LIN {X 0,Y 432.341,Z 505.628,A -85,B 0,C 180,E1 -9485.631,E2 -9485.631} C_VEL
LIN {X 0,Y 432.351,Z 505.616,A -85,B 0,C 180,E1 -9489.341,E2 -9489.341} C_VEL
LIN {X 0,Y 432.331,Z 505.631,A -85,B 0,C 180,E1 -9491.796,E2 -9491.796} C_VEL
LIN {X 0,Y 432.338,Z 505.625,A -85,B 0,C 180,E1 -9494.345,E2 -9494.345} C_VEL
LIN {X 0,Y 432.315,Z 505.635,A -85,B 0,C 180,E1 -9497.015,E2 -9497.015} C_VEL
LIN {X 0,Y 432.35,Z 505.628,A -85,B 0,C 180,E1 -9499.817,E2 -9499.817} C_VEL
LIN {X 0,Y 432.31,Z 505.629,A -85,B 0,C 180,E1 -9503.022,E2 -9503.022} C_VEL
LIN {X 0,Y 432.353,Z 505.626,A -85,B 0,C 180,E1 -9505.996,E2 -9505.996} C_VEL
LIN {X 0,Y 432.388,Z 505.616,A -85,B 0,C 180,E1 -9509.744,E2 -9509.744} C_VEL
LIN {X 0,Y 432.392,Z 505.622,A -85,B 0,C 180,E1 -9513.372,E2 -9513.372} C_VEL
LIN {X 0,Y 432.363,Z 505.611,A -85,B 0,C 180,E1 -9516.023,E2 -9516.023} C_VEL
LIN {X 0,Y 432.342,Z 505.631,A -85,B 0,C 180,E1 -9519.046,E2 -9519.046} C_VEL
LIN {X 0,Y 432.369,Z 505.617,A -85,B 0,C 180,E1 -9522.011,E2 -9522.011} C_VEL
LIN {X 0,Y 432.386,Z 505.615,A -85,B 0,C 180,E1 -9524.926,E2 -9524.926} C_VEL
LIN {X 0,Y 432.472,Z 505.611,A -85,B 0,C 180,E1 -9527.804,E2 -9527.804} C_VEL
LIN {X 0,Y 432.483,Z 505.597,A -85,B 0,C 180,E1 -9531.59,E2 -9531.59} C_VEL
LIN {X 0,Y 432.595,Z 505.593,A -85,B 0,C 180,E1 -9534.406,E2 -9534.406} C_VEL
LIN {X 0,Y 432.597,Z 505.59,A -85,B 0,C 180,E1 -9538.138,E2 -9538.138} C_VEL
LIN {X 0,Y 432.725,Z 505.562,A -85,B 0,C 180,E1 -9540,E2 -9540} C_VEL
LIN {X 0,Y 432.599,Z 505.594,A -85,B 0,C 180,E1 -9542.794,E2 -9542.794} C_VEL
LIN {X 0,Y 432.568,Z 505.597,A -85,B 0,C 180,E1 -9546.531,E2 -9546.531} C_VEL
LIN {X 0,Y 432.435,Z 505.61,A -85,B 0,C 180,E1 -9549.354,E2 -9549.354} C_VEL
LIN {X 0,Y 432.422,Z 505.621,A -85,B 0,C 180,E1 -9552.804,E2 -9552.804} C_VEL
LIN {X 0,Y 432.404,Z 505.607,A -85,B 0,C 180,E1 -9556.479,E2 -9556.479} C_VEL
LIN {X 0,Y 432.331,Z 505.629,A -85,B 0,C 180,E1 -9559.961,E2 -9559.961} C_VEL
LIN {X 0,Y 432.312,Z 505.625,A -85,B 0,C 180,E1 -9562.965,E2 -9562.965} C_VEL
LIN {X 0,Y 432.358,Z 505.625,A -85,B 0,C 180,E1 -9566.033,E2 -9566.033} C_VEL
LIN {X 0,Y 432.347,Z 505.622,A -85,B 0,C 180,E1 -9569.188,E2 -9569.188} C_VEL
LIN {X 0,Y 432.327,Z 505.63,A -85,B 0,C 180,E1 -9572.296,E2 -9572.296} C_VEL
LIN {X 0,Y 432.336,Z 505.627,A -85,B 0,C 180,E1 -9574.678,E2 -9574.678} C_VEL
LIN {X 0,Y 432.343,Z 505.629,A -85,B 0,C 180,E1 -9578.15,E2 -9578.15} C_VEL
LIN {X 0,Y 432.33,Z 505.633,A -85,B 0,C 180,E1 -9581.603,E2 -9581.603} C_VEL
LIN {X 0,Y 432.339,Z 505.628,A -85,B 0,C 180,E1 -9584.347,E2 -9584.347} C_VEL
LIN {X 0,Y 432.324,Z 505.633,A -85,B 0,C 180,E1 -9587.016,E2 -9587.016} C_VEL
LIN {X 0,Y 432.336,Z 505.628,A -85,B 0,C 180,E1 -9589.821,E2 -9589.821} C_VEL
LIN {X 0,Y 432.306,Z 505.639,A -85,B 0,C 180,E1 -9593.023,E2 -9593.023} C_VEL
LIN {X 0,Y 432.36,Z 505.626,A -85,B 0,C 180,E1 -9595.997,E2 -9595.997} C_VEL
LIN {X 0,Y 432.349,Z 505.63,A -85,B 0,C 180,E1 -9599.49,E2 -9599.49} C_VEL
LIN {X 0,Y 432.453,Z 505.772,A -85,B 0,C 180,E1 -9601.948,E2 -9601.948} C_VEL
LIN {X 0,Y 434.883,Z 517.9,A -85,B 0,C 180,E1 -9604.318,E2 -9604.318} C_VEL
LIN {X 0,Y 435.122,Z 522.494,A -85,B 0,C 180,E1 -9605.169,E2 -9605.169} C_VEL
LIN {X 0,Y 434.407,Z 540.816,A -85,B 0,C 180,E1 -9608.405,E2 -9608.405} C_VEL
LIN {X 0,Y 434.177,Z 547.705,A -85,B 0,C 180,E1 -9609.575,E2 -9609.575} C_VEL
LIN {X 0,Y 437.623,Z 566.618,A -85,B 0,C 180,E1 -9610.058,E2 -9610.058} C_VEL
LIN {X 0,Y 436.607,Z 656.61,A -85,B 0,C 180,E1 -9611.565,E2 -9611.565} C_VEL
LIN {X 0,Y 436.236,Z 669.411,A -85,B 0,C 180,E1 -9611.944,E2 -9611.944} C_VEL
LIN {X 0,Y 435.822,Z 682.12,A -85,B 0,C 180,E1 -9612.522,E2 -9612.522} C_VEL
LIN {X 0,Y 435.249,Z 693.577,A -85,B 0,C 180,E1 -9613.225,E2 -9613.225} C_VEL
LIN {X 0,Y 434.972,Z 698.627,A -85,B 0,C 180,E1 -9613.597,E2 -9613.597} C_VEL
LIN {X 0,Y 434.086,Z 703.686,A -85,B 0,C 180,E1 -9613.987,E2 -9613.987} C_VEL
LIN {X 0,Y 430.753,Z 711.627,A -85,B 0,C 180,E1 -9614.639,E2 -9614.639} C_VEL
LIN {X 0,Y 427.364,Z 719.148,A -85,B 0,C 180,E1 -9615.375,E2 -9615.375} C_VEL
LIN {X 0,Y 426.383,Z 723.435,A -85,B 0,C 180,E1 -9615.901,E2 -9615.901} C_VEL
LIN {X 0,Y 425.771,Z 732.739,A -85,B 0,C 180,E1 -9617.298,E2 -9617.298} C_VEL
LIN {X 0,Y 425.345,Z 739.588,A -85,B 0,C 180,E1 -9618.564,E2 -9618.564} C_VEL
LIN {X 0,Y 424.83,Z 745.924,A -85,B 0,C 180,E1 -9619.997,E2 -9619.997} C_VEL
LIN {X 0,Y 424.555,Z 750.93,A -85,B 0,C 180,E1 -9621.432,E2 -9621.432} C_VEL
LIN {X 0,Y 424.34,Z 754.79,A -85,B 0,C 180,E1 -9622.865,E2 -9622.865} C_VEL
LIN {X 0,Y 424.233,Z 757.622,A -85,B 0,C 180,E1 -9624.296,E2 -9624.296} C_VEL
LIN {X 0,Y 424.166,Z 758.957,A -85,B 0,C 180,E1 -9625.248,E2 -9625.248} C_VEL
LIN {X 0,Y 424.159,Z 760.464,A -85,B 0,C 180,E1 -9627.151,E2 -9627.151} C_VEL
LIN {X 0,Y 424.145,Z 760.612,A -85,B 0,C 180,E1 -9628.101,E2 -9628.101} C_VEL
LIN {X 0,Y 424.087,Z 759.718,A -85,B 0,C 180,E1 -9630,E2 -9630} C_VEL
LIN {X 0,Y 424.102,Z 758.7,A -85,B 0,C 180,E1 -9630.949,E2 -9630.949} C_VEL
LIN {X 0,Y 424.219,Z 757.234,A -85,B 0,C 180,E1 -9631.899,E2 -9631.899} C_VEL
LIN {X 0,Y 424.418,Z 754.261,A -85,B 0,C 180,E1 -9633.322,E2 -9633.322} C_VEL
LIN {X 0,Y 424.52,Z 750.254,A -85,B 0,C 180,E1 -9634.748,E2 -9634.748} C_VEL
LIN {X 0,Y 424.845,Z 745.088,A -85,B 0,C 180,E1 -9636.173,E2 -9636.173} C_VEL
LIN {X 0,Y 425.293,Z 738.607,A -85,B 0,C 180,E1 -9637.597,E2 -9637.597} C_VEL
LIN {X 0,Y 425.786,Z 730.565,A -85,B 0,C 180,E1 -9639.021,E2 -9639.021} C_VEL
LIN {X 0,Y 426.388,Z 722.292,A -85,B 0,C 180,E1 -9640.206,E2 -9640.206} C_VEL
LIN {X 0,Y 427.118,Z 712.126,A -85,B 0,C 180,E1 -9641.388,E2 -9641.388} C_VEL
LIN {X 0,Y 427.639,Z 702.118,A -85,B 0,C 180,E1 -9642.336,E2 -9642.336} C_VEL
LIN {X 0,Y 428.303,Z 691.197,A -85,B 0,C 180,E1 -9643.16,E2 -9643.16} C_VEL
LIN {X 0,Y 428.945,Z 678.921,A -85,B 0,C 180,E1 -9643.864,E2 -9643.864} C_VEL
LIN {X 0,Y 429.327,Z 666.008,A -85,B 0,C 180,E1 -9644.402,E2 -9644.402} C_VEL
LIN {X 0,Y 429.593,Z 653.002,A -85,B 0,C 180,E1 -9644.744,E2 -9644.744} C_VEL
LIN {X 0,Y 430.444,Z 566.841,A -85,B 0,C 180,E1 -9646.19,E2 -9646.19} C_VEL
LIN {X 0,Y 427.125,Z 547.784,A -85,B 0,C 180,E1 -9646.673,E2 -9646.673} C_VEL
LIN {X 0,Y 427.683,Z 530.472,A -85,B 0,C 180,E1 -9649.686,E2 -9649.686} C_VEL
LIN {X 0,Y 428.1,Z 520.701,A -85,B 0,C 180,E1 -9651.424,E2 -9651.424} C_VEL
LIN {X 0,Y 425.367,Z 506.508,A -85,B 0,C 180,E1 -9654.201,E2 -9654.201} C_VEL
LIN {X 0,Y 425.351,Z 506.503,A -85,B 0,C 180,E1 -9657.557,E2 -9657.557} C_VEL
LIN {X 0,Y 425.289,Z 506.512,A -85,B 0,C 180,E1 -9660.815,E2 -9660.815} C_VEL
LIN {X 0,Y 425.312,Z 506.503,A -85,B 0,C 180,E1 -9664.287,E2 -9664.287} C_VEL
LIN {X 0,Y 425.278,Z 506.508,A -85,B 0,C 180,E1 -9667.693,E2 -9667.693} C_VEL
LIN {X 0,Y 425.279,Z 506.505,A -85,B 0,C 180,E1 -9670.519,E2 -9670.519} C_VEL
LIN {X 0,Y 425.314,Z 506.504,A -85,B 0,C 180,E1 -9673.358,E2 -9673.358} C_VEL
LIN {X 0,Y 425.262,Z 506.508,A -85,B 0,C 180,E1 -9676.647,E2 -9676.647} C_VEL
LIN {X 0,Y 425.287,Z 506.507,A -85,B 0,C 180,E1 -9679.872,E2 -9679.872} C_VEL
LIN {X 0,Y 425.281,Z 506.512,A -85,B 0,C 180,E1 -9682.486,E2 -9682.486} C_VEL
LIN {X 0,Y 425.335,Z 506.683,A -85,B 0,C 180,E1 -9685.491,E2 -9685.491} C_VEL
LIN {X 0,Y 430.311,Z 521.652,A -85,B 0,C 180,E1 -9685.987,E2 -9685.987} C_VEL
LIN {X 0,Y 429.49,Z 582.153,A -85,B 0,C 180,E1 -9687.13,E2 -9687.13} C_VEL
LIN {X 0,Y 429.057,Z 613.843,A -85,B 0,C 180,E1 -9687.748,E2 -9687.748} C_VEL
LIN {X 0,Y 428.746,Z 627.654,A -85,B 0,C 180,E1 -9688.224,E2 -9688.224} C_VEL
LIN {X 0,Y 428.311,Z 640.607,A -85,B 0,C 180,E1 -9688.885,E2 -9688.885} C_VEL
LIN {X 0,Y 427.76,Z 652.022,A -85,B 0,C 180,E1 -9689.654,E2 -9689.654} C_VEL
LIN {X 0,Y 427.225,Z 662.724,A -85,B 0,C 180,E1 -9690.563,E2 -9690.563} C_VEL
LIN {X 0,Y 426.642,Z 673.648,A -85,B 0,C 180,E1 -9691.732,E2 -9691.732} C_VEL
LIN {X 0,Y 426.074,Z 682.949,A -85,B 0,C 180,E1 -9692.961,E2 -9692.961} C_VEL
LIN {X 0,Y 425.558,Z 691.253,A -85,B 0,C 180,E1 -9694.309,E2 -9694.309} C_VEL
LIN {X 0,Y 425.147,Z 698.777,A -85,B 0,C 180,E1 -9695.849,E2 -9695.849} C_VEL
LIN {X 0,Y 424.86,Z 703.791,A -85,B 0,C 180,E1 -9697.124,E2 -9697.124} C_VEL
LIN {X 0,Y 424.617,Z 708.497,A -85,B 0,C 180,E1 -9698.646,E2 -9698.646} C_VEL
LIN {X 0,Y 424.485,Z 710.957,A -85,B 0,C 180,E1 -9699.654,E2 -9699.654} C_VEL
LIN {X 0,Y 424.356,Z 712.969,A -85,B 0,C 180,E1 -9700.732,E2 -9700.732} C_VEL
LIN {X 0,Y 424.283,Z 714.276,A -85,B 0,C 180,E1 -9701.656,E2 -9701.656} C_VEL
LIN {X 0,Y 424.247,Z 715.261,A -85,B 0,C 180,E1 -9702.651,E2 -9702.651} C_VEL
LIN {X 0,Y 424.261,Z 715.804,A -85,B 0,C 180,E1 -9703.897,E2 -9703.897} C_VEL
LIN {X 0,Y 424.267,Z 715.456,A -85,B 0,C 180,E1 -9705.612,E2 -9705.612} C_VEL
LIN {X 0,Y 424.341,Z 714.619,A -85,B 0,C 180,E1 -9706.593,E2 -9706.593} C_VEL
LIN {X 0,Y 424.458,Z 713.231,A -85,B 0,C 180,E1 -9707.654,E2 -9707.654} C_VEL
LIN {X 0,Y 424.647,Z 710.624,A -85,B 0,C 180,E1 -9709.028,E2 -9709.028} C_VEL
LIN {X 0,Y 424.888,Z 706.828,A -85,B 0,C 180,E1 -9710.479,E2 -9710.479} C_VEL
LIN {X 0,Y 425.242,Z 701.869,A -85,B 0,C 180,E1 -9711.924,E2 -9711.924} C_VEL
LIN {X 0,Y 425.661,Z 695.613,A -85,B 0,C 180,E1 -9713.363,E2 -9713.363} C_VEL
LIN {X 0,Y 426.188,Z 687.757,A -85,B 0,C 180,E1 -9714.796,E2 -9714.796} C_VEL
LIN {X 0,Y 426.711,Z 679.77,A -85,B 0,C 180,E1 -9715.986,E2 -9715.986} C_VEL
LIN {X 0,Y 427.38,Z 670.015,A -85,B 0,C 180,E1 -9717.172,E2 -9717.172} C_VEL
LIN {X 0,Y 427.998,Z 660.441,A -85,B 0,C 180,E1 -9718.118,E2 -9718.118} C_VEL
LIN {X 0,Y 428.622,Z 648.437,A -85,B 0,C 180,E1 -9719.06,E2 -9719.06} C_VEL
LIN {X 0,Y 429.185,Z 635.524,A -85,B 0,C 180,E1 -9719.834,E2 -9719.834} C_VEL
LIN {X 0,Y 429.552,Z 622.759,A -85,B 0,C 180,E1 -9720.381,E2 -9720.381} C_VEL
LIN {X 0,Y 429.765,Z 609.087,A -85,B 0,C 180,E1 -9720.761,E2 -9720.761} C_VEL
LIN {X 0,Y 431.395,Z 523.126,A -85,B 0,C 180,E1 -9722.451,E2 -9722.451} C_VEL
LIN {X 0,Y 426.079,Z 509.418,A -85,B 0,C 180,E1 -9723.073,E2 -9723.073} C_VEL
LIN {X 0,Y 425.34,Z 506.506,A -85,B 0,C 180,E1 -9724.027,E2 -9724.027} C_VEL
LIN {X 0,Y 425.57,Z 506.477,A -85,B 0,C 180,E1 -9725.686,E2 -9725.686} C_VEL
LIN {X 0,Y 425.434,Z 506.492,A -85,B 0,C 180,E1 -9728.55,E2 -9728.55} C_VEL
LIN {X 0,Y 425.423,Z 506.491,A -85,B 0,C 180,E1 -9732.401,E2 -9732.401} C_VEL
LIN {X 0,Y 425.379,Z 506.497,A -85,B 0,C 180,E1 -9736.312,E2 -9736.312} C_VEL
LIN {X 0,Y 425.32,Z 506.504,A -85,B 0,C 180,E1 -9739.636,E2 -9739.636} C_VEL
LIN {X 0,Y 425.299,Z 506.508,A -85,B 0,C 180,E1 -9743.365,E2 -9743.365} C_VEL
LIN {X 0,Y 425.341,Z 506.502,A -85,B 0,C 180,E1 -9746.845,E2 -9746.845} C_VEL
LIN {X 0,Y 425.311,Z 506.501,A -85,B 0,C 180,E1 -9749.718,E2 -9749.718} C_VEL
LIN {X 0,Y 425.276,Z 506.511,A -85,B 0,C 180,E1 -9753.049,E2 -9753.049} C_VEL
LIN {X 0,Y 425.278,Z 506.505,A -85,B 0,C 180,E1 -9755.93,E2 -9755.93} C_VEL
LIN {X 0,Y 425.296,Z 506.511,A -85,B 0,C 180,E1 -9759.045,E2 -9759.045} C_VEL
LIN {X 0,Y 425.27,Z 506.511,A -85,B 0,C 180,E1 -9762.654,E2 -9762.654} C_VEL
LIN {X 0,Y 425.264,Z 506.511,A -85,B 0,C 180,E1 -9766.046,E2 -9766.046} C_VEL
LIN {X 0,Y 425.272,Z 506.515,A -85,B 0,C 180,E1 -9768.622,E2 -9768.622} C_VEL
LIN {X 0,Y 425.31,Z 506.509,A -85,B 0,C 180,E1 -9771.104,E2 -9771.104} C_VEL
LIN {X 0,Y 425.298,Z 506.511,A -85,B 0,C 180,E1 -9774.665,E2 -9774.665} C_VEL
LIN {X 0,Y 425.264,Z 506.517,A -85,B 0,C 180,E1 -9778.074,E2 -9778.074} C_VEL
LIN {X 0,Y 425.327,Z 506.527,A -85,B 0,C 180,E1 -9780.148,E2 -9780.148} C_VEL
LIN {X 0,Y 428.003,Z 518.179,A -85,B 0,C 180,E1 -9782.628,E2 -9782.628} C_VEL
LIN {X 0,Y 429.122,Z 525.624,A -85,B 0,C 180,E1 -9784.103,E2 -9784.103} C_VEL
LIN {X 0,Y 427.797,Z 544.959,A -85,B 0,C 180,E1 -9787.56,E2 -9787.56} C_VEL
LIN {X 0,Y 426.59,Z 564.666,A -85,B 0,C 180,E1 -9790.977,E2 -9790.977} C_VEL
LIN {X 0,Y 429.519,Z 585.448,A -85,B 0,C 180,E1 -9791.571,E2 -9791.571} C_VEL
LIN {X 0,Y 430.567,Z 596.351,A -85,B 0,C 180,E1 -9791.848,E2 -9791.848} C_VEL
LIN {X 0,Y 429.24,Z 676.045,A -85,B 0,C 180,E1 -9793.411,E2 -9793.411} C_VEL
LIN {X 0,Y 428.636,Z 691.691,A -85,B 0,C 180,E1 -9793.938,E2 -9793.938} C_VEL
LIN {X 0,Y 428.13,Z 703.871,A -85,B 0,C 180,E1 -9794.468,E2 -9794.468} C_VEL
LIN {X 0,Y 427.45,Z 716.668,A -85,B 0,C 180,E1 -9795.236,E2 -9795.236} C_VEL
LIN {X 0,Y 426.867,Z 727.179,A -85,B 0,C 180,E1 -9796.059,E2 -9796.059} C_VEL
LIN {X 0,Y 426.279,Z 736.997,A -85,B 0,C 180,E1 -9797.019,E2 -9797.019} C_VEL
LIN {X 0,Y 425.715,Z 745.975,A -85,B 0,C 180,E1 -9798.091,E2 -9798.091} C_VEL
LIN {X 0,Y 425.098,Z 755.69,A -85,B 0,C 180,E1 -9799.522,E2 -9799.522} C_VEL
LIN {X 0,Y 424.699,Z 763.401,A -85,B 0,C 180,E1 -9800.955,E2 -9800.955} C_VEL
LIN {X 0,Y 424.43,Z 769.564,A -85,B 0,C 180,E1 -9802.388,E2 -9802.388} C_VEL
LIN {X 0,Y 424.271,Z 773.978,A -85,B 0,C 180,E1 -9803.666,E2 -9803.666} C_VEL
LIN {X 0,Y 424.237,Z 778.164,A -85,B 0,C 180,E1 -9805.249,E2 -9805.249} C_VEL
LIN {X 0,Y 424.125,Z 780.078,A -85,B 0,C 180,E1 -9806.2,E2 -9806.2} C_VEL
LIN {X 0,Y 424.212,Z 781.549,A -85,B 0,C 180,E1 -9807.151,E2 -9807.151} C_VEL
LIN {X 0,Y 424.176,Z 782.574,A -85,B 0,C 180,E1 -9808.101,E2 -9808.101} C_VEL
LIN {X 0,Y 424.096,Z 783.448,A -85,B 0,C 180,E1 -9810,E2 -9810} C_VEL
LIN {X 0,Y 424.099,Z 783.253,A -85,B 0,C 180,E1 -9810.95,E2 -9810.95} C_VEL
LIN {X 0,Y 424.176,Z 782.654,A -85,B 0,C 180,E1 -9811.899,E2 -9811.899} C_VEL
LIN {X 0,Y 424.214,Z 781.661,A -85,B 0,C 180,E1 -9812.849,E2 -9812.849} C_VEL
LIN {X 0,Y 424.128,Z 780.257,A -85,B 0,C 180,E1 -9813.8,E2 -9813.8} C_VEL
LIN {X 0,Y 424.258,Z 777.312,A -85,B 0,C 180,E1 -9815.227,E2 -9815.227} C_VEL
LIN {X 0,Y 424.307,Z 773.307,A -85,B 0,C 180,E1 -9816.658,E2 -9816.658} C_VEL
LIN {X 0,Y 424.577,Z 767.111,A -85,B 0,C 180,E1 -9818.328,E2 -9818.328} C_VEL
LIN {X 0,Y 424.939,Z 760.348,A -85,B 0,C 180,E1 -9819.76,E2 -9819.76} C_VEL
LIN {X 0,Y 425.342,Z 753.443,A -85,B 0,C 180,E1 -9820.953,E2 -9820.953} C_VEL
LIN {X 0,Y 425.907,Z 745.112,A -85,B 0,C 180,E1 -9822.145,E2 -9822.145} C_VEL
LIN {X 0,Y 426.582,Z 734.805,A -85,B 0,C 180,E1 -9823.335,E2 -9823.335} C_VEL
LIN {X 0,Y 427.179,Z 724.581,A -85,B 0,C 180,E1 -9824.287,E2 -9824.287} C_VEL
LIN {X 0,Y 427.86,Z 713.375,A -85,B 0,C 180,E1 -9825.115,E2 -9825.115} C_VEL
LIN {X 0,Y 428.404,Z 701.928,A -85,B 0,C 180,E1 -9825.766,E2 -9825.766} C_VEL
LIN {X 0,Y 428.967,Z 688.747,A -85,B 0,C 180,E1 -9826.294,E2 -9826.294} C_VEL
LIN {X 0,Y 429.312,Z 675.9,A -85,B 0,C 180,E1 -9826.616,E2 -9826.616} C_VEL
LIN {X 0,Y 429.987,Z 593.708,A -85,B 0,C 180,E1 -9828.001,E2 -9828.001} C_VEL
LIN {X 0,Y 426.519,Z 567.791,A -85,B 0,C 180,E1 -9828.616,E2 -9828.616} C_VEL
LIN {X 0,Y 427.528,Z 549.649,A -85,B 0,C 180,E1 -9831.707,E2 -9831.707} C_VEL
LIN {X 0,Y 428.717,Z 530.735,A -85,B 0,C 180,E1 -9834.968,E2 -9834.968} C_VEL
LIN {X 0,Y 429.071,Z 525.356,A -85,B 0,C 180,E1 -9835.906,E2 -9835.906} C_VEL
LIN {X 0,Y 427.368,Z 515.912,A -85,B 0,C 180,E1 -9837.681,E2 -9837.681} C_VEL
LIN {X 0,Y 425.317,Z 506.508,A -85,B 0,C 180,E1 -9839.508,E2 -9839.508} C_VEL
LIN {X 0,Y 425.28,Z 506.513,A -85,B 0,C 180,E1 -9843.047,E2 -9843.047} C_VEL
LIN {X 0,Y 425.279,Z 506.505,A -85,B 0,C 180,E1 -9845.928,E2 -9845.928} C_VEL
LIN {X 0,Y 425.297,Z 506.489,A -85,B 0,C 180,E1 -9849.043,E2 -9849.043} C_VEL
LIN {X 0,Y 425.275,Z 506.51,A -85,B 0,C 180,E1 -9852.652,E2 -9852.652} C_VEL
LIN {X 0,Y 425.256,Z 506.512,A -85,B 0,C 180,E1 -9856.043,E2 -9856.043} C_VEL
LIN {X 0,Y 425.299,Z 506.499,A -85,B 0,C 180,E1 -9858.624,E2 -9858.624} C_VEL
LIN {X 0,Y 425.317,Z 506.509,A -85,B 0,C 180,E1 -9861.103,E2 -9861.103} C_VEL
LIN {X 0,Y 425.294,Z 506.502,A -85,B 0,C 180,E1 -9864.664,E2 -9864.664} C_VEL
LIN {X 0,Y 425.259,Z 506.505,A -85,B 0,C 180,E1 -9868.073,E2 -9868.073} C_VEL
LIN {X 0,Y 425.33,Z 506.505,A -85,B 0,C 180,E1 -9871.368,E2 -9871.368} C_VEL
LIN {X 0,Y 425.288,Z 506.504,A -85,B 0,C 180,E1 -9874.554,E2 -9874.554} C_VEL
LIN {X 0,Y 425.279,Z 506.506,A -85,B 0,C 180,E1 -9877.661,E2 -9877.661} C_VEL
LIN {X 0,Y 425.353,Z 506.499,A -85,B 0,C 180,E1 -9880.704,E2 -9880.704} C_VEL
LIN {X 0,Y 425.379,Z 506.483,A -85,B 0,C 180,E1 -9883.688,E2 -9883.688} C_VEL
LIN {X 0,Y 425.421,Z 506.491,A -85,B 0,C 180,E1 -9887.599,E2 -9887.599} C_VEL
LIN {X 0,Y 425.434,Z 506.474,A -85,B 0,C 180,E1 -9891.45,E2 -9891.45} C_VEL
LIN {X 0,Y 425.57,Z 506.468,A -85,B 0,C 180,E1 -9894.314,E2 -9894.314} C_VEL
LIN {X 0,Y 425.566,Z 506.466,A -85,B 0,C 180,E1 -9898.107,E2 -9898.107} C_VEL
LIN {X 0,Y 425.695,Z 506.437,A -85,B 0,C 180,E1 -9900,E2 -9900} C_VEL
LIN {X 0,Y 425.551,Z 506.473,A -85,B 0,C 180,E1 -9902.84,E2 -9902.84} C_VEL
LIN {X 0,Y 425.57,Z 506.469,A -85,B 0,C 180,E1 -9905.687,E2 -9905.687} C_VEL
LIN {X 0,Y 425.434,Z 506.474,A -85,B 0,C 180,E1 -9908.551,E2 -9908.551} C_VEL
LIN {X 0,Y 425.404,Z 506.492,A -85,B 0,C 180,E1 -9912.402,E2 -9912.402} C_VEL
LIN {X 0,Y 425.38,Z 506.48,A -85,B 0,C 180,E1 -9916.312,E2 -9916.312} C_VEL
LIN {X 0,Y 425.321,Z 506.503,A -85,B 0,C 180,E1 -9919.636,E2 -9919.636} C_VEL
LIN {X 0,Y 425.3,Z 506.497,A -85,B 0,C 180,E1 -9923.366,E2 -9923.366} C_VEL
LIN {X 0,Y 425.343,Z 506.504,A -85,B 0,C 180,E1 -9926.845,E2 -9926.845} C_VEL
LIN {X 0,Y 425.313,Z 506.496,A -85,B 0,C 180,E1 -9929.718,E2 -9929.718} C_VEL
LIN {X 0,Y 425.28,Z 506.512,A -85,B 0,C 180,E1 -9933.049,E2 -9933.049} C_VEL
LIN {X 0,Y 425.28,Z 506.506,A -85,B 0,C 180,E1 -9935.93,E2 -9935.93} C_VEL
LIN {X 0,Y 425.297,Z 506.507,A -85,B 0,C 180,E1 -9939.045,E2 -9939.045} C_VEL
LIN {X 0,Y 425.275,Z 506.514,A -85,B 0,C 180,E1 -9942.654,E2 -9942.654} C_VEL
LIN {X 0,Y 425.268,Z 506.51,A -85,B 0,C 180,E1 -9946.046,E2 -9946.046} C_VEL
LIN {X 0,Y 425.275,Z 506.512,A -85,B 0,C 180,E1 -9948.623,E2 -9948.623} C_VEL
LIN {X 0,Y 425.309,Z 506.508,A -85,B 0,C 180,E1 -9951.104,E2 -9951.104} C_VEL
LIN {X 0,Y 425.299,Z 506.503,A -85,B 0,C 180,E1 -9954.665,E2 -9954.665} C_VEL
LIN {X 0,Y 425.266,Z 506.505,A -85,B 0,C 180,E1 -9958.074,E2 -9958.074} C_VEL
LIN {X 0,Y 425.394,Z 506.602,A -85,B 0,C 180,E1 -9961.676,E2 -9961.676} C_VEL
LIN {X 0,Y 427.979,Z 519.202,A -85,B 0,C 180,E1 -9964.168,E2 -9964.168} C_VEL
LIN {X 0,Y 428.246,Z 523.672,A -85,B 0,C 180,E1 -9965.003,E2 -9965.003} C_VEL
LIN {X 0,Y 427.496,Z 542.181,A -85,B 0,C 180,E1 -9968.291,E2 -9968.291} C_VEL
LIN {X 0,Y 427.293,Z 547.849,A -85,B 0,C 180,E1 -9969.257,E2 -9969.257} C_VEL
LIN {X 0,Y 430.922,Z 567.646,A -85,B 0,C 180,E1 -9969.773,E2 -9969.773} C_VEL
LIN {X 0,Y 429.842,Z 656.668,A -85,B 0,C 180,E1 -9971.285,E2 -9971.285} C_VEL
LIN {X 0,Y 429.433,Z 670.008,A -85,B 0,C 180,E1 -9971.687,E2 -9971.687} C_VEL
LIN {X 0,Y 428.982,Z 682.969,A -85,B 0,C 180,E1 -9972.296,E2 -9972.296} C_VEL
LIN {X 0,Y 428.356,Z 695.136,A -85,B 0,C 180,E1 -9973.069,E2 -9973.069} C_VEL
LIN {X 0,Y 427.592,Z 706.643,A -85,B 0,C 180,E1 -9974.02,E2 -9974.02} C_VEL
LIN {X 0,Y 426.87,Z 716.94,A -85,B 0,C 180,E1 -9975.093,E2 -9975.093} C_VEL
LIN {X 0,Y 426.383,Z 723.435,A -85,B 0,C 180,E1 -9975.901,E2 -9975.901} C_VEL
LIN {X 0,Y 425.44,Z 727.581,A -85,B 0,C 180,E1 -9976.457,E2 -9976.457} C_VEL
LIN {X 0,Y 422.156,Z 733.954,A -85,B 0,C 180,E1 -9977.389,E2 -9977.389} C_VEL
LIN {X 0,Y 418.909,Z 739.728,A -85,B 0,C 180,E1 -9978.399,E2 -9978.399} C_VEL
LIN {X 0,Y 418.033,Z 742.893,A -85,B 0,C 180,E1 -9979.068,E2 -9979.068} C_VEL
LIN {X 0,Y 417.67,Z 747.817,A -85,B 0,C 180,E1 -9980.313,E2 -9980.313} C_VEL
LIN {X 0,Y 417.414,Z 752.45,A -85,B 0,C 180,E1 -9981.772,E2 -9981.772} C_VEL
LIN {X 0,Y 417.234,Z 755.972,A -85,B 0,C 180,E1 -9983.229,E2 -9983.229} C_VEL
LIN {X 0,Y 417.151,Z 757.779,A -85,B 0,C 180,E1 -9984.198,E2 -9984.198} C_VEL
LIN {X 0,Y 417.098,Z 759.122,A -85,B 0,C 180,E1 -9985.167,E2 -9985.167} C_VEL
LIN {X 0,Y 417.056,Z 760.644,A -85,B 0,C 180,E1 -9987.102,E2 -9987.102} C_VEL
LIN {X 0,Y 417.072,Z 760.806,A -85,B 0,C 180,E1 -9988.069,E2 -9988.069} C_VEL
LIN {X 0,Y 417.007,Z 759.926,A -85,B 0,C 180,E1 -9990,E2 -9990} C_VEL
LIN {X 0,Y 417.025,Z 758.916,A -85,B 0,C 180,E1 -9990.966,E2 -9990.966} C_VEL
LIN {X 0,Y 417.146,Z 757.464,A -85,B 0,C 180,E1 -9991.931,E2 -9991.931} C_VEL
LIN {X 0,Y 417.354,Z 754.505,A -85,B 0,C 180,E1 -9993.379,E2 -9993.379} C_VEL
LIN {X 0,Y 417.446,Z 750.513,A -85,B 0,C 180,E1 -9994.829,E2 -9994.829} C_VEL
LIN {X 0,Y 417.809,Z 745.363,A -85,B 0,C 180,E1 -9996.277,E2 -9996.277} C_VEL
LIN {X 0,Y 418.345,Z 737.704,A -85,B 0,C 180,E1 -9997.966,E2 -9997.966} C_VEL
LIN {X 0,Y 418.897,Z 729.333,A -85,B 0,C 180,E1 -9999.414,E2 -9999.414} C_VEL
LIN {X 0,Y 419.556,Z 720.757,A -85,B 0,C 180,E1 -10000.618,E2 -10000.618} C_VEL
LIN {X 0,Y 420.282,Z 710.241,A -85,B 0,C 180,E1 -10001.82,E2 -10001.82} C_VEL
LIN {X 0,Y 420.973,Z 699.672,A -85,B 0,C 180,E1 -10002.779,E2 -10002.779} C_VEL
LIN {X 0,Y 421.585,Z 687.961,A -85,B 0,C 180,E1 -10003.619,E2 -10003.619} C_VEL
LIN {X 0,Y 422.247,Z 675.854,A -85,B 0,C 180,E1 -10004.273,E2 -10004.273} C_VEL
LIN {X 0,Y 422.57,Z 663.566,A -85,B 0,C 180,E1 -10004.745,E2 -10004.745} C_VEL
LIN {X 0,Y 422.84,Z 650.096,A -85,B 0,C 180,E1 -10005.061,E2 -10005.061} C_VEL
LIN {X 0,Y 423.713,Z 568.069,A -85,B 0,C 180,E1 -10006.456,E2 -10006.456} C_VEL
LIN {X 0,Y 420.228,Z 547.953,A -85,B 0,C 180,E1 -10006.971,E2 -10006.971} C_VEL
LIN {X 0,Y 420.799,Z 530.532,A -85,B 0,C 180,E1 -10010.022,E2 -10010.022} C_VEL
LIN {X 0,Y 421.198,Z 522.122,A -85,B 0,C 180,E1 -10011.535,E2 -10011.535} C_VEL
LIN {X 0,Y 418.331,Z 507.385,A -85,B 0,C 180,E1 -10014.437,E2 -10014.437} C_VEL
LIN {X 0,Y 418.293,Z 507.38,A -85,B 0,C 180,E1 -10018.062,E2 -10018.062} C_VEL
LIN {X 0,Y 418.213,Z 507.393,A -85,B 0,C 180,E1 -10021.395,E2 -10021.395} C_VEL
LIN {X 0,Y 418.266,Z 507.383,A -85,B 0,C 180,E1 -10024.579,E2 -10024.579} C_VEL
LIN {X 0,Y 418.227,Z 507.386,A -85,B 0,C 180,E1 -10027.832,E2 -10027.832} C_VEL
LIN {X 0,Y 418.259,Z 507.381,A -85,B 0,C 180,E1 -10030.942,E2 -10030.942} C_VEL
LIN {X 0,Y 418.266,Z 507.38,A -85,B 0,C 180,E1 -10033.737,E2 -10033.737} C_VEL
LIN {X 0,Y 418.214,Z 507.384,A -85,B 0,C 180,E1 -10036.449,E2 -10036.449} C_VEL
LIN {X 0,Y 418.221,Z 507.391,A -85,B 0,C 180,E1 -10039.129,E2 -10039.129} C_VEL
LIN {X 0,Y 418.231,Z 507.388,A -85,B 0,C 180,E1 -10042.164,E2 -10042.164} C_VEL
LIN {X 0,Y 418.287,Z 507.384,A -85,B 0,C 180,E1 -10045.2,E2 -10045.2} C_VEL
LIN {X 0,Y 423.551,Z 522.9,A -85,B 0,C 180,E1 -10045.743,E2 -10045.743} C_VEL
LIN {X 0,Y 422.186,Z 613.794,A -85,B 0,C 180,E1 -10047.512,E2 -10047.512} C_VEL
LIN {X 0,Y 421.861,Z 627.602,A -85,B 0,C 180,E1 -10047.989,E2 -10047.989} C_VEL
LIN {X 0,Y 421.416,Z 640.677,A -85,B 0,C 180,E1 -10048.658,E2 -10048.658} C_VEL
LIN {X 0,Y 420.809,Z 653.187,A -85,B 0,C 180,E1 -10049.516,E2 -10049.516} C_VEL
LIN {X 0,Y 420.194,Z 664.482,A -85,B 0,C 180,E1 -10050.513,E2 -10050.513} C_VEL
LIN {X 0,Y 419.571,Z 675.648,A -85,B 0,C 180,E1 -10051.757,E2 -10051.757} C_VEL
LIN {X 0,Y 418.976,Z 685.096,A -85,B 0,C 180,E1 -10053.069,E2 -10053.069} C_VEL
LIN {X 0,Y 418.461,Z 692.861,A -85,B 0,C 180,E1 -10054.402,E2 -10054.402} C_VEL
LIN {X 0,Y 418.057,Z 700.09,A -85,B 0,C 180,E1 -10055.941,E2 -10055.941} C_VEL
LIN {X 0,Y 417.776,Z 704.958,A -85,B 0,C 180,E1 -10057.237,E2 -10057.237} C_VEL
LIN {X 0,Y 417.538,Z 709.532,A -85,B 0,C 180,E1 -10058.783,E2 -10058.783} C_VEL
LIN {X 0,Y 417.316,Z 713.287,A -85,B 0,C 180,E1 -10060.574,E2 -10060.574} C_VEL
LIN {X 0,Y 417.177,Z 715.535,A -85,B 0,C 180,E1 -10062.347,E2 -10062.347} C_VEL
LIN {X 0,Y 417.182,Z 716.327,A -85,B 0,C 180,E1 -10063.785,E2 -10063.785} C_VEL
LIN {X 0,Y 417.178,Z 716.155,A -85,B 0,C 180,E1 -10065.362,E2 -10065.362} C_VEL
LIN {X 0,Y 417.244,Z 715.494,A -85,B 0,C 180,E1 -10066.36,E2 -10066.36} C_VEL
LIN {X 0,Y 417.373,Z 714.027,A -85,B 0,C 180,E1 -10067.586,E2 -10067.586} C_VEL
LIN {X 0,Y 417.627,Z 710.775,A -85,B 0,C 180,E1 -10069.332,E2 -10069.332} C_VEL
LIN {X 0,Y 417.93,Z 706.838,A -85,B 0,C 180,E1 -10070.807,E2 -10070.807} C_VEL
LIN {X 0,Y 418.326,Z 701.257,A -85,B 0,C 180,E1 -10072.391,E2 -10072.391} C_VEL
LIN {X 0,Y 418.897,Z 694.025,A -85,B 0,C 180,E1 -10073.981,E2 -10073.981} C_VEL
LIN {X 0,Y 419.492,Z 685.694,A -85,B 0,C 180,E1 -10075.435,E2 -10075.435} C_VEL
LIN {X 0,Y 420.109,Z 677.096,A -85,B 0,C 180,E1 -10076.643,E2 -10076.643} C_VEL
LIN {X 0,Y 420.776,Z 666.556,A -85,B 0,C 180,E1 -10077.846,E2 -10077.846} C_VEL
LIN {X 0,Y 421.477,Z 656.037,A -85,B 0,C 180,E1 -10078.805,E2 -10078.805} C_VEL
LIN {X 0,Y 422.118,Z 644.082,A -85,B 0,C 180,E1 -10079.659,E2 -10079.659} C_VEL
LIN {X 0,Y 422.614,Z 631.175,A -85,B 0,C 180,E1 -10080.357,E2 -10080.357} C_VEL
LIN {X 0,Y 422.97,Z 618.582,A -85,B 0,C 180,E1 -10080.833,E2 -10080.833} C_VEL
LIN {X 0,Y 423.232,Z 600.594,A -85,B 0,C 180,E1 -10081.245,E2 -10081.245} C_VEL
LIN {X 0,Y 424.78,Z 524.585,A -85,B 0,C 180,E1 -10082.789,E2 -10082.789} C_VEL
LIN {X 0,Y 419.862,Z 512.396,A -85,B 0,C 180,E1 -10083.35,E2 -10083.35} C_VEL
LIN {X 0,Y 418.95,Z 510.164,A -85,B 0,C 180,E1 -10083.486,E2 -10083.486} C_VEL
LIN {X 0,Y 418.33,Z 507.378,A -85,B 0,C 180,E1 -10084.396,E2 -10084.396} C_VEL
LIN {X 0,Y 418.487,Z 507.359,A -85,B 0,C 180,E1 -10086.751,E2 -10086.751} C_VEL
LIN {X 0,Y 418.352,Z 507.375,A -85,B 0,C 180,E1 -10089.671,E2 -10089.671} C_VEL
LIN {X 0,Y 418.347,Z 507.376,A -85,B 0,C 180,E1 -10093.007,E2 -10093.007} C_VEL
LIN {X 0,Y 418.304,Z 507.379,A -85,B 0,C 180,E1 -10096.736,E2 -10096.736} C_VEL
LIN {X 0,Y 418.262,Z 507.383,A -85,B 0,C 180,E1 -10099.791,E2 -10099.791} C_VEL
LIN {X 0,Y 418.23,Z 507.389,A -85,B 0,C 180,E1 -10102.737,E2 -10102.737} C_VEL
LIN {X 0,Y 418.263,Z 507.38,A -85,B 0,C 180,E1 -10105.904,E2 -10105.904} C_VEL
LIN {X 0,Y 418.267,Z 507.382,A -85,B 0,C 180,E1 -10109.162,E2 -10109.162} C_VEL
LIN {X 0,Y 418.251,Z 507.384,A -85,B 0,C 180,E1 -10112.845,E2 -10112.845} C_VEL
LIN {X 0,Y 418.242,Z 507.381,A -85,B 0,C 180,E1 -10116.239,E2 -10116.239} C_VEL
LIN {X 0,Y 418.247,Z 507.384,A -85,B 0,C 180,E1 -10119.682,E2 -10119.682} C_VEL
LIN {X 0,Y 418.224,Z 507.387,A -85,B 0,C 180,E1 -10122.322,E2 -10122.322} C_VEL
LIN {X 0,Y 418.235,Z 507.39,A -85,B 0,C 180,E1 -10125.11,E2 -10125.11} C_VEL
LIN {X 0,Y 418.238,Z 507.388,A -85,B 0,C 180,E1 -10127.768,E2 -10127.768} C_VEL
LIN {X 0,Y 418.254,Z 507.387,A -85,B 0,C 180,E1 -10130.619,E2 -10130.619} C_VEL
LIN {X 0,Y 418.243,Z 507.386,A -85,B 0,C 180,E1 -10133.977,E2 -10133.977} C_VEL
LIN {X 0,Y 418.256,Z 507.392,A -85,B 0,C 180,E1 -10137.157,E2 -10137.157} C_VEL
LIN {X 0,Y 418.279,Z 507.471,A -85,B 0,C 180,E1 -10139.764,E2 -10139.764} C_VEL
LIN {X 0,Y 421.127,Z 519.704,A -85,B 0,C 180,E1 -10142.446,E2 -10142.446} C_VEL
LIN {X 0,Y 422.26,Z 527.343,A -85,B 0,C 180,E1 -10143.996,E2 -10143.996} C_VEL
LIN {X 0,Y 420.891,Z 546.092,A -85,B 0,C 180,E1 -10147.416,E2 -10147.416} C_VEL
LIN {X 0,Y 419.722,Z 563.932,A -85,B 0,C 180,E1 -10150.581,E2 -10150.581} C_VEL
LIN {X 0,Y 422.658,Z 584.437,A -85,B 0,C 180,E1 -10151.192,E2 -10151.192} C_VEL
LIN {X 0,Y 423.906,Z 597.069,A -85,B 0,C 180,E1 -10151.533,E2 -10151.533} C_VEL
LIN {X 0,Y 422.474,Z 675.292,A -85,B 0,C 180,E1 -10153.107,E2 -10153.107} C_VEL
LIN {X 0,Y 421.864,Z 689.198,A -85,B 0,C 180,E1 -10153.58,E2 -10153.58} C_VEL
LIN {X 0,Y 421.267,Z 703.487,A -85,B 0,C 180,E1 -10154.209,E2 -10154.209} C_VEL
LIN {X 0,Y 420.552,Z 716.323,A -85,B 0,C 180,E1 -10154.988,E2 -10154.988} C_VEL
LIN {X 0,Y 419.936,Z 726.926,A -85,B 0,C 180,E1 -10155.829,E2 -10155.829} C_VEL
LIN {X 0,Y 419.254,Z 737.78,A -85,B 0,C 180,E1 -10156.921,E2 -10156.921} C_VEL
LIN {X 0,Y 418.613,Z 747.488,A -85,B 0,C 180,E1 -10158.132,E2 -10158.132} C_VEL
LIN {X 0,Y 418.076,Z 755.43,A -85,B 0,C 180,E1 -10159.344,E2 -10159.344} C_VEL
LIN {X 0,Y 417.637,Z 763.158,A -85,B 0,C 180,E1 -10160.801,E2 -10160.801} C_VEL
LIN {X 0,Y 417.364,Z 769.331,A -85,B 0,C 180,E1 -10162.258,E2 -10162.258} C_VEL
LIN {X 0,Y 417.192,Z 774.099,A -85,B 0,C 180,E1 -10163.675,E2 -10163.675} C_VEL
LIN {X 0,Y 417.167,Z 777.949,A -85,B 0,C 180,E1 -10165.168,E2 -10165.168} C_VEL
LIN {X 0,Y 417.04,Z 779.867,A -85,B 0,C 180,E1 -10166.135,E2 -10166.135} C_VEL
LIN {X 0,Y 417.105,Z 781.345,A -85,B 0,C 180,E1 -10167.103,E2 -10167.103} C_VEL
LIN {X 0,Y 417.102,Z 782.375,A -85,B 0,C 180,E1 -10168.069,E2 -10168.069} C_VEL
LIN {X 0,Y 417.015,Z 783.256,A -85,B 0,C 180,E1 -10170,E2 -10170} C_VEL
LIN {X 0,Y 417.021,Z 783.069,A -85,B 0,C 180,E1 -10170.966,E2 -10170.966} C_VEL
LIN {X 0,Y 417.103,Z 782.473,A -85,B 0,C 180,E1 -10171.931,E2 -10171.931} C_VEL
LIN {X 0,Y 417.107,Z 781.483,A -85,B 0,C 180,E1 -10172.897,E2 -10172.897} C_VEL
LIN {X 0,Y 417.042,Z 780.086,A -85,B 0,C 180,E1 -10173.865,E2 -10173.865} C_VEL
LIN {X 0,Y 417.172,Z 777.148,A -85,B 0,C 180,E1 -10175.316,E2 -10175.316} C_VEL
LIN {X 0,Y 417.242,Z 773.153,A -85,B 0,C 180,E1 -10176.771,E2 -10176.771} C_VEL
LIN {X 0,Y 417.516,Z 766.97,A -85,B 0,C 180,E1 -10178.47,E2 -10178.47} C_VEL
LIN {X 0,Y 417.9,Z 760.219,A -85,B 0,C 180,E1 -10179.926,E2 -10179.926} C_VEL
LIN {X 0,Y 418.436,Z 751.806,A -85,B 0,C 180,E1 -10181.382,E2 -10181.382} C_VEL
LIN {X 0,Y 419.092,Z 743.117,A -85,B 0,C 180,E1 -10182.592,E2 -10182.592} C_VEL
LIN {X 0,Y 419.743,Z 733.245,A -85,B 0,C 180,E1 -10183.714,E2 -10183.714} C_VEL
LIN {X 0,Y 420.392,Z 723.129,A -85,B 0,C 180,E1 -10184.646,E2 -10184.646} C_VEL
LIN {X 0,Y 421.095,Z 711.535,A -85,B 0,C 180,E1 -10185.488,E2 -10185.488} C_VEL
LIN {X 0,Y 421.741,Z 699.46,A -85,B 0,C 180,E1 -10186.146,E2 -10186.146} C_VEL
LIN {X 0,Y 422.248,Z 687.175,A -85,B 0,C 180,E1 -10186.623,E2 -10186.623} C_VEL
LIN {X 0,Y 422.566,Z 674.858,A -85,B 0,C 180,E1 -10186.921,E2 -10186.921} C_VEL
LIN {X 0,Y 423.296,Z 594.707,A -85,B 0,C 180,E1 -10188.289,E2 -10188.289} C_VEL
LIN {X 0,Y 419.553,Z 566.858,A -85,B 0,C 180,E1 -10188.982,E2 -10188.982} C_VEL
LIN {X 0,Y 420.633,Z 548.987,A -85,B 0,C 180,E1 -10192.081,E2 -10192.081} C_VEL
LIN {X 0,Y 421.867,Z 530.076,A -85,B 0,C 180,E1 -10195.402,E2 -10195.402} C_VEL
LIN {X 0,Y 421.978,Z 525.197,A -85,B 0,C 180,E1 -10196.276,E2 -10196.276} C_VEL
LIN {X 0,Y 419.3,Z 512.132,A -85,B 0,C 180,E1 -10198.808,E2 -10198.808} C_VEL
LIN {X 0,Y 418.278,Z 507.384,A -85,B 0,C 180,E1 -10199.782,E2 -10199.782} C_VEL
LIN {X 0,Y 418.246,Z 507.387,A -85,B 0,C 180,E1 -10203.676,E2 -10203.676} C_VEL
LIN {X 0,Y 418.237,Z 507.368,A -85,B 0,C 180,E1 -10207.223,E2 -10207.223} C_VEL
LIN {X 0,Y 418.251,Z 507.378,A -85,B 0,C 180,E1 -10209.681,E2 -10209.681} C_VEL
LIN {X 0,Y 418.229,Z 507.387,A -85,B 0,C 180,E1 -10212.321,E2 -10212.321} C_VEL
LIN {X 0,Y 418.234,Z 507.388,A -85,B 0,C 180,E1 -10215.108,E2 -10215.108} C_VEL
LIN {X 0,Y 418.251,Z 507.377,A -85,B 0,C 180,E1 -10217.768,E2 -10217.768} C_VEL
LIN {X 0,Y 418.262,Z 507.383,A -85,B 0,C 180,E1 -10220.616,E2 -10220.616} C_VEL
LIN {X 0,Y 418.24,Z 507.379,A -85,B 0,C 180,E1 -10223.976,E2 -10223.976} C_VEL
LIN {X 0,Y 418.251,Z 507.386,A -85,B 0,C 180,E1 -10227.155,E2 -10227.155} C_VEL
LIN {X 0,Y 418.267,Z 507.377,A -85,B 0,C 180,E1 -10230.838,E2 -10230.838} C_VEL
LIN {X 0,Y 418.263,Z 507.377,A -85,B 0,C 180,E1 -10234.096,E2 -10234.096} C_VEL
LIN {X 0,Y 418.224,Z 507.381,A -85,B 0,C 180,E1 -10237.263,E2 -10237.263} C_VEL
LIN {X 0,Y 418.275,Z 507.379,A -85,B 0,C 180,E1 -10240.364,E2 -10240.364} C_VEL
LIN {X 0,Y 418.308,Z 507.363,A -85,B 0,C 180,E1 -10243.404,E2 -10243.404} C_VEL
LIN {X 0,Y 418.346,Z 507.374,A -85,B 0,C 180,E1 -10246.994,E2 -10246.994} C_VEL
LIN {X 0,Y 418.352,Z 507.363,A -85,B 0,C 180,E1 -10250.329,E2 -10250.329} C_VEL
LIN {X 0,Y 418.487,Z 507.348,A -85,B 0,C 180,E1 -10253.249,E2 -10253.249} C_VEL
LIN {X 0,Y 418.338,Z 507.377,A -85,B 0,C 180,E1 -10255.182,E2 -10255.182} C_VEL
LIN {X 0,Y 418.536,Z 507.342,A -85,B 0,C 180,E1 -10258.076,E2 -10258.076} C_VEL
LIN {X 0,Y 418.665,Z 507.312,A -85,B 0,C 180,E1 -10260,E2 -10260} C_VEL
LIN {X 0,Y 418.504,Z 507.351,A -85,B 0,C 180,E1 -10262.888,E2 -10262.888} C_VEL
LIN {X 0,Y 418.485,Z 507.351,A -85,B 0,C 180,E1 -10266.611,E2 -10266.611} C_VEL
LIN {X 0,Y 418.334,Z 507.367,A -85,B 0,C 180,E1 -10269.672,E2 -10269.672} C_VEL
LIN {X 0,Y 418.338,Z 507.378,A -85,B 0,C 180,E1 -10273.001,E2 -10273.001} C_VEL
LIN {X 0,Y 418.305,Z 507.363,A -85,B 0,C 180,E1 -10276.736,E2 -10276.736} C_VEL
LIN {X 0,Y 418.263,Z 507.382,A -85,B 0,C 180,E1 -10279.791,E2 -10279.791} C_VEL
LIN {X 0,Y 418.231,Z 507.38,A -85,B 0,C 180,E1 -10282.737,E2 -10282.737} C_VEL
LIN {X 0,Y 418.265,Z 507.381,A -85,B 0,C 180,E1 -10285.905,E2 -10285.905} C_VEL
LIN {X 0,Y 418.269,Z 507.375,A -85,B 0,C 180,E1 -10289.162,E2 -10289.162} C_VEL
LIN {X 0,Y 418.256,Z 507.388,A -85,B 0,C 180,E1 -10292.846,E2 -10292.846} C_VEL
LIN {X 0,Y 418.244,Z 507.383,A -85,B 0,C 180,E1 -10296.24,E2 -10296.24} C_VEL
LIN {X 0,Y 418.248,Z 507.382,A -85,B 0,C 180,E1 -10299.683,E2 -10299.683} C_VEL
LIN {X 0,Y 418.229,Z 507.39,A -85,B 0,C 180,E1 -10302.322,E2 -10302.322} C_VEL
LIN {X 0,Y 418.241,Z 507.392,A -85,B 0,C 180,E1 -10305.111,E2 -10305.111} C_VEL
LIN {X 0,Y 418.241,Z 507.385,A -85,B 0,C 180,E1 -10307.768,E2 -10307.768} C_VEL
LIN {X 0,Y 418.255,Z 507.385,A -85,B 0,C 180,E1 -10310.62,E2 -10310.62} C_VEL
LIN {X 0,Y 418.243,Z 507.384,A -85,B 0,C 180,E1 -10313.977,E2 -10313.977} C_VEL
LIN {X 0,Y 418.258,Z 507.383,A -85,B 0,C 180,E1 -10317.157,E2 -10317.157} C_VEL
LIN {X 0,Y 418.27,Z 507.384,A -85,B 0,C 180,E1 -10320.896,E2 -10320.896} C_VEL
LIN {X 0,Y 418.313,Z 507.474,A -85,B 0,C 180,E1 -10321.392,E2 -10321.392} C_VEL
LIN {X 0,Y 421.055,Z 520.566,A -85,B 0,C 180,E1 -10324.015,E2 -10324.015} C_VEL
LIN {X 0,Y 421.364,Z 524.865,A -85,B 0,C 180,E1 -10324.83,E2 -10324.83} C_VEL
LIN {X 0,Y 420.6,Z 543.59,A -85,B 0,C 180,E1 -10328.175,E2 -10328.175} C_VEL
LIN {X 0,Y 420.426,Z 547.914,A -85,B 0,C 180,E1 -10328.918,E2 -10328.918} C_VEL
LIN {X 0,Y 424.212,Z 568.754,A -85,B 0,C 180,E1 -10329.479,E2 -10329.479} C_VEL
LIN {X 0,Y 423.065,Z 657.159,A -85,B 0,C 180,E1 -10331.005,E2 -10331.005} C_VEL
LIN {X 0,Y 422.655,Z 670.49,A -85,B 0,C 180,E1 -10331.418,E2 -10331.418} C_VEL
LIN {X 0,Y 422.211,Z 682.779,A -85,B 0,C 180,E1 -10332.004,E2 -10332.004} C_VEL
LIN {X 0,Y 421.556,Z 695.01,A -85,B 0,C 180,E1 -10332.788,E2 -10332.788} C_VEL
LIN {X 0,Y 420.744,Z 706.601,A -85,B 0,C 180,E1 -10333.753,E2 -10333.753} C_VEL
LIN {X 0,Y 419.984,Z 716.938,A -85,B 0,C 180,E1 -10334.843,E2 -10334.843} C_VEL
LIN {X 0,Y 419.191,Z 727.12,A -85,B 0,C 180,E1 -10336.178,E2 -10336.178} C_VEL
LIN {X 0,Y 418.633,Z 735.927,A -85,B 0,C 180,E1 -10337.641,E2 -10337.641} C_VEL
LIN {X 0,Y 418.033,Z 742.893,A -85,B 0,C 180,E1 -10339.068,E2 -10339.068} C_VEL
LIN {X 0,Y 417.167,Z 745.876,A -85,B 0,C 180,E1 -10339.758,E2 -10339.758} C_VEL
LIN {X 0,Y 414,Z 750.231,A -85,B 0,C 180,E1 -10340.909,E2 -10340.909} C_VEL
LIN {X 0,Y 410.907,Z 753.848,A -85,B 0,C 180,E1 -10342.122,E2 -10342.122} C_VEL
LIN {X 0,Y 410.173,Z 755.675,A -85,B 0,C 180,E1 -10342.902,E2 -10342.902} C_VEL
LIN {X 0,Y 410.071,Z 757.935,A -85,B 0,C 180,E1 -10344.098,E2 -10344.098} C_VEL
LIN {X 0,Y 410.032,Z 759.289,A -85,B 0,C 180,E1 -10345.084,E2 -10345.084} C_VEL
LIN {X 0,Y 409.953,Z 760.825,A -85,B 0,C 180,E1 -10347.052,E2 -10347.052} C_VEL
LIN {X 0,Y 410.001,Z 760.999,A -85,B 0,C 180,E1 -10348.035,E2 -10348.035} C_VEL
LIN {X 0,Y 409.929,Z 760.134,A -85,B 0,C 180,E1 -10350,E2 -10350} C_VEL
LIN {X 0,Y 409.95,Z 759.131,A -85,B 0,C 180,E1 -10350.982,E2 -10350.982} C_VEL
LIN {X 0,Y 410.076,Z 757.692,A -85,B 0,C 180,E1 -10351.964,E2 -10351.964} C_VEL
LIN {X 0,Y 410.29,Z 754.747,A -85,B 0,C 180,E1 -10353.437,E2 -10353.437} C_VEL
LIN {X 0,Y 410.377,Z 750.772,A -85,B 0,C 180,E1 -10354.912,E2 -10354.912} C_VEL
LIN {X 0,Y 410.776,Z 745.637,A -85,B 0,C 180,E1 -10356.385,E2 -10356.385} C_VEL
LIN {X 0,Y 411.228,Z 739.193,A -85,B 0,C 180,E1 -10357.858,E2 -10357.858} C_VEL
LIN {X 0,Y 411.814,Z 731.19,A -85,B 0,C 180,E1 -10359.33,E2 -10359.33} C_VEL
LIN {X 0,Y 412.461,Z 722.984,A -85,B 0,C 180,E1 -10360.554,E2 -10360.554} C_VEL
LIN {X 0,Y 413.242,Z 712.881,A -85,B 0,C 180,E1 -10361.776,E2 -10361.776} C_VEL
LIN {X 0,Y 413.979,Z 701.576,A -85,B 0,C 180,E1 -10362.874,E2 -10362.874} C_VEL
LIN {X 0,Y 414.591,Z 690.334,A -85,B 0,C 180,E1 -10363.728,E2 -10363.728} C_VEL
LIN {X 0,Y 415.347,Z 677.655,A -85,B 0,C 180,E1 -10364.452,E2 -10364.452} C_VEL
LIN {X 0,Y 415.739,Z 665.402,A -85,B 0,C 180,E1 -10364.96,E2 -10364.96} C_VEL
LIN {X 0,Y 416.005,Z 652.018,A -85,B 0,C 180,E1 -10365.303,E2 -10365.303} C_VEL
LIN {X 0,Y 416.956,Z 569.162,A -85,B 0,C 180,E1 -10366.733,E2 -10366.733} C_VEL
LIN {X 0,Y 413.332,Z 548.042,A -85,B 0,C 180,E1 -10367.29,E2 -10367.29} C_VEL
LIN {X 0,Y 413.941,Z 530.622,A -85,B 0,C 180,E1 -10370.368,E2 -10370.368} C_VEL
LIN {X 0,Y 414.305,Z 523.693,A -85,B 0,C 180,E1 -10371.624,E2 -10371.624} C_VEL
LIN {X 0,Y 411.504,Z 509.363,A -85,B 0,C 180,E1 -10374.446,E2 -10374.446} C_VEL
LIN {X 0,Y 411.248,Z 508.267,A -85,B 0,C 180,E1 -10374.711,E2 -10374.711} C_VEL
LIN {X 0,Y 411.261,Z 508.257,A -85,B 0,C 180,E1 -10377.477,E2 -10377.477} C_VEL
LIN {X 0,Y 411.191,Z 508.268,A -85,B 0,C 180,E1 -10380.847,E2 -10380.847} C_VEL
LIN {X 0,Y 411.206,Z 508.26,A -85,B 0,C 180,E1 -10384.333,E2 -10384.333} C_VEL
LIN {X 0,Y 411.194,Z 508.263,A -85,B 0,C 180,E1 -10387.973,E2 -10387.973} C_VEL
LIN {X 0,Y 411.2,Z 508.263,A -85,B 0,C 180,E1 -10391.233,E2 -10391.233} C_VEL
LIN {X 0,Y 411.223,Z 508.257,A -85,B 0,C 180,E1 -10394.483,E2 -10394.483} C_VEL
LIN {X 0,Y 411.176,Z 508.265,A -85,B 0,C 180,E1 -10398.194,E2 -10398.194} C_VEL
LIN {X 0,Y 411.218,Z 508.265,A -85,B 0,C 180,E1 -10400.775,E2 -10400.775} C_VEL
LIN {X 0,Y 411.2,Z 508.266,A -85,B 0,C 180,E1 -10404.471,E2 -10404.471} C_VEL
LIN {X 0,Y 411.209,Z 508.271,A -85,B 0,C 180,E1 -10404.931,E2 -10404.931} C_VEL
LIN {X 0,Y 416.832,Z 524.767,A -85,B 0,C 180,E1 -10405.509,E2 -10405.509} C_VEL
LIN {X 0,Y 415.3,Z 614.49,A -85,B 0,C 180,E1 -10407.289,E2 -10407.289} C_VEL
LIN {X 0,Y 414.962,Z 628.169,A -85,B 0,C 180,E1 -10407.772,E2 -10407.772} C_VEL
LIN {X 0,Y 414.516,Z 640.93,A -85,B 0,C 180,E1 -10408.434,E2 -10408.434} C_VEL
LIN {X 0,Y 413.93,Z 652.603,A -85,B 0,C 180,E1 -10409.237,E2 -10409.237} C_VEL
LIN {X 0,Y 413.321,Z 663.915,A -85,B 0,C 180,E1 -10410.226,E2 -10410.226} C_VEL
LIN {X 0,Y 412.703,Z 674.42,A -85,B 0,C 180,E1 -10411.383,E2 -10411.383} C_VEL
LIN {X 0,Y 412.126,Z 683.321,A -85,B 0,C 180,E1 -10412.585,E2 -10412.585} C_VEL
LIN {X 0,Y 411.58,Z 691.417,A -85,B 0,C 180,E1 -10413.915,E2 -10413.915} C_VEL
LIN {X 0,Y 411.154,Z 698.517,A -85,B 0,C 180,E1 -10415.351,E2 -10415.351} C_VEL
LIN {X 0,Y 410.791,Z 704.348,A -85,B 0,C 180,E1 -10416.827,E2 -10416.827} C_VEL
LIN {X 0,Y 410.544,Z 709.197,A -85,B 0,C 180,E1 -10418.404,E2 -10418.404} C_VEL
LIN {X 0,Y 410.293,Z 712.775,A -85,B 0,C 180,E1 -10419.965,E2 -10419.965} C_VEL
LIN {X 0,Y 410.198,Z 714.537,A -85,B 0,C 180,E1 -10421.002,E2 -10421.002} C_VEL
LIN {X 0,Y 410.12,Z 715.797,A -85,B 0,C 180,E1 -10422.033,E2 -10422.033} C_VEL
LIN {X 0,Y 410.119,Z 716.847,A -85,B 0,C 180,E1 -10423.662,E2 -10423.662} C_VEL
LIN {X 0,Y 410.093,Z 716.855,A -85,B 0,C 180,E1 -10425.104,E2 -10425.104} C_VEL
LIN {X 0,Y 410.157,Z 716.302,A -85,B 0,C 180,E1 -10426.12,E2 -10426.12} C_VEL
LIN {X 0,Y 410.319,Z 714.868,A -85,B 0,C 180,E1 -10427.496,E2 -10427.496} C_VEL
LIN {X 0,Y 410.545,Z 712.024,A -85,B 0,C 180,E1 -10429.146,E2 -10429.146} C_VEL
LIN {X 0,Y 410.852,Z 708.313,A -85,B 0,C 180,E1 -10430.647,E2 -10430.647} C_VEL
LIN {X 0,Y 411.282,Z 702.726,A -85,B 0,C 180,E1 -10432.342,E2 -10432.342} C_VEL
LIN {X 0,Y 411.83,Z 696.126,A -85,B 0,C 180,E1 -10433.877,E2 -10433.877} C_VEL
LIN {X 0,Y 412.459,Z 688.114,A -85,B 0,C 180,E1 -10435.357,E2 -10435.357} C_VEL
LIN {X 0,Y 413.069,Z 679.94,A -85,B 0,C 180,E1 -10436.586,E2 -10436.586} C_VEL
LIN {X 0,Y 413.779,Z 669.953,A -85,B 0,C 180,E1 -10437.81,E2 -10437.81} C_VEL
LIN {X 0,Y 414.497,Z 660.072,A -85,B 0,C 180,E1 -10438.785,E2 -10438.785} C_VEL
LIN {X 0,Y 415.166,Z 649.169,A -85,B 0,C 180,E1 -10439.652,E2 -10439.652} C_VEL
LIN {X 0,Y 415.732,Z 636.714,A -85,B 0,C 180,E1 -10440.424,E2 -10440.424} C_VEL
LIN {X 0,Y 416.154,Z 623.743,A -85,B 0,C 180,E1 -10440.998,E2 -10440.998} C_VEL
LIN {X 0,Y 416.421,Z 610.13,A -85,B 0,C 180,E1 -10441.39,E2 -10441.39} C_VEL
LIN {X 0,Y 418.219,Z 526.322,A -85,B 0,C 180,E1 -10443.131,E2 -10443.131} C_VEL
LIN {X 0,Y 413.779,Z 515.328,A -85,B 0,C 180,E1 -10443.666,E2 -10443.666} C_VEL
LIN {X 0,Y 411.817,Z 510.944,A -85,B 0,C 180,E1 -10443.914,E2 -10443.914} C_VEL
LIN {X 0,Y 411.292,Z 508.254,A -85,B 0,C 180,E1 -10444.778,E2 -10444.778} C_VEL
LIN {X 0,Y 411.454,Z 508.236,A -85,B 0,C 180,E1 -10446.867,E2 -10446.867} C_VEL
LIN {X 0,Y 411.3,Z 508.253,A -85,B 0,C 180,E1 -10449.838,E2 -10449.838} C_VEL
LIN {X 0,Y 411.305,Z 508.254,A -85,B 0,C 180,E1 -10453.109,E2 -10453.109} C_VEL
LIN {X 0,Y 411.249,Z 508.258,A -85,B 0,C 180,E1 -10456.889,E2 -10456.889} C_VEL
LIN {X 0,Y 411.222,Z 508.259,A -85,B 0,C 180,E1 -10459.987,E2 -10459.987} C_VEL
LIN {X 0,Y 411.195,Z 508.266,A -85,B 0,C 180,E1 -10463.148,E2 -10463.148} C_VEL
LIN {X 0,Y 411.23,Z 508.257,A -85,B 0,C 180,E1 -10466.381,E2 -10466.381} C_VEL
LIN {X 0,Y 411.204,Z 508.258,A -85,B 0,C 180,E1 -10469.712,E2 -10469.712} C_VEL
LIN {X 0,Y 411.2,Z 508.263,A -85,B 0,C 180,E1 -10473.156,E2 -10473.156} C_VEL
LIN {X 0,Y 411.189,Z 508.262,A -85,B 0,C 180,E1 -10476.554,E2 -10476.554} C_VEL
LIN {X 0,Y 411.211,Z 508.26,A -85,B 0,C 180,E1 -10479.729,E2 -10479.729} C_VEL
LIN {X 0,Y 411.168,Z 508.271,A -85,B 0,C 180,E1 -10483.134,E2 -10483.134} C_VEL
LIN {X 0,Y 411.168,Z 508.268,A -85,B 0,C 180,E1 -10485.881,E2 -10485.881} C_VEL
LIN {X 0,Y 411.161,Z 508.272,A -85,B 0,C 180,E1 -10488.772,E2 -10488.772} C_VEL
LIN {X 0,Y 411.197,Z 508.264,A -85,B 0,C 180,E1 -10492.028,E2 -10492.028} C_VEL
LIN {X 0,Y 411.204,Z 508.266,A -85,B 0,C 180,E1 -10495.667,E2 -10495.667} C_VEL
LIN {X 0,Y 411.231,Z 508.366,A -85,B 0,C 180,E1 -10499.335,E2 -10499.335} C_VEL
LIN {X 0,Y 413.577,Z 518.215,A -85,B 0,C 180,E1 -10501.589,E2 -10501.589} C_VEL
LIN {X 0,Y 415.2,Z 526.415,A -85,B 0,C 180,E1 -10503.348,E2 -10503.348} C_VEL
LIN {X 0,Y 415.276,Z 530.59,A -85,B 0,C 180,E1 -10504.165,E2 -10504.165} C_VEL
LIN {X 0,Y 413.828,Z 548.733,A -85,B 0,C 180,E1 -10507.536,E2 -10507.536} C_VEL
LIN {X 0,Y 412.858,Z 563.479,A -85,B 0,C 180,E1 -10510.175,E2 -10510.175} C_VEL
LIN {X 0,Y 415.937,Z 583.832,A -85,B 0,C 180,E1 -10510.814,E2 -10510.814} C_VEL
LIN {X 0,Y 417.282,Z 597.784,A -85,B 0,C 180,E1 -10511.197,E2 -10511.197} C_VEL
LIN {X 0,Y 415.745,Z 674.719,A -85,B 0,C 180,E1 -10512.793,E2 -10512.793} C_VEL
LIN {X 0,Y 415.136,Z 688.533,A -85,B 0,C 180,E1 -10513.274,E2 -10513.274} C_VEL
LIN {X 0,Y 414.326,Z 705.344,A -85,B 0,C 180,E1 -10514.063,E2 -10514.063} C_VEL
LIN {X 0,Y 413.577,Z 717.68,A -85,B 0,C 180,E1 -10514.855,E2 -10514.855} C_VEL
LIN {X 0,Y 412.91,Z 728.471,A -85,B 0,C 180,E1 -10515.762,E2 -10515.762} C_VEL
LIN {X 0,Y 412.23,Z 738.558,A -85,B 0,C 180,E1 -10516.819,E2 -10516.819} C_VEL
LIN {X 0,Y 411.633,Z 747.214,A -85,B 0,C 180,E1 -10517.928,E2 -10517.928} C_VEL
LIN {X 0,Y 411.063,Z 755.169,A -85,B 0,C 180,E1 -10519.16,E2 -10519.16} C_VEL
LIN {X 0,Y 410.6,Z 762.914,A -85,B 0,C 180,E1 -10520.642,E2 -10520.642} C_VEL
LIN {X 0,Y 410.297,Z 769.097,A -85,B 0,C 180,E1 -10522.124,E2 -10522.124} C_VEL
LIN {X 0,Y 410.112,Z 774.225,A -85,B 0,C 180,E1 -10523.687,E2 -10523.687} C_VEL
LIN {X 0,Y 410.074,Z 777.732,A -85,B 0,C 180,E1 -10525.084,E2 -10525.084} C_VEL
LIN {X 0,Y 409.959,Z 779.655,A -85,B 0,C 180,E1 -10526.068,E2 -10526.068} C_VEL
LIN {X 0,Y 410,Z 781.14,A -85,B 0,C 180,E1 -10527.052,E2 -10527.052} C_VEL
LIN {X 0,Y 410.03,Z 782.175,A -85,B 0,C 180,E1 -10528.036,E2 -10528.036} C_VEL
LIN {X 0,Y 409.937,Z 783.064,A -85,B 0,C 180,E1 -10530,E2 -10530} C_VEL
LIN {X 0,Y 409.946,Z 782.884,A -85,B 0,C 180,E1 -10530.982,E2 -10530.982} C_VEL
LIN {X 0,Y 410.03,Z 782.292,A -85,B 0,C 180,E1 -10531.964,E2 -10531.964} C_VEL
LIN {X 0,Y 410.001,Z 781.305,A -85,B 0,C 180,E1 -10532.948,E2 -10532.948} C_VEL
LIN {X 0,Y 409.961,Z 779.915,A -85,B 0,C 180,E1 -10533.932,E2 -10533.932} C_VEL
LIN {X 0,Y 410.069,Z 776.984,A -85,B 0,C 180,E1 -10535.409,E2 -10535.409} C_VEL
LIN {X 0,Y 410.178,Z 773,A -85,B 0,C 180,E1 -10536.888,E2 -10536.888} C_VEL
LIN {X 0,Y 410.467,Z 766.831,A -85,B 0,C 180,E1 -10538.616,E2 -10538.616} C_VEL
LIN {X 0,Y 410.882,Z 760.093,A -85,B 0,C 180,E1 -10540.097,E2 -10540.097} C_VEL
LIN {X 0,Y 411.465,Z 751.702,A -85,B 0,C 180,E1 -10541.577,E2 -10541.577} C_VEL
LIN {X 0,Y 412.132,Z 743.032,A -85,B 0,C 180,E1 -10542.808,E2 -10542.808} C_VEL
LIN {X 0,Y 412.882,Z 732.578,A -85,B 0,C 180,E1 -10544.012,E2 -10544.012} C_VEL
LIN {X 0,Y 413.623,Z 721.64,A -85,B 0,C 180,E1 -10545.017,E2 -10545.017} C_VEL
LIN {X 0,Y 414.382,Z 709.599,A -85,B 0,C 180,E1 -10545.871,E2 -10545.871} C_VEL
LIN {X 0,Y 415.077,Z 696.998,A -85,B 0,C 180,E1 -10546.538,E2 -10546.538} C_VEL
LIN {X 0,Y 415.583,Z 684.433,A -85,B 0,C 180,E1 -10546.992,E2 -10546.992} C_VEL
LIN {X 0,Y 415.886,Z 670.211,A -85,B 0,C 180,E1 -10547.296,E2 -10547.296} C_VEL
LIN {X 0,Y 416.592,Z 595.599,A -85,B 0,C 180,E1 -10548.59,E2 -10548.59} C_VEL
LIN {X 0,Y 412.649,Z 566.008,A -85,B 0,C 180,E1 -10549.338,E2 -10549.338} C_VEL
LIN {X 0,Y 413.71,Z 548.289,A -85,B 0,C 180,E1 -10552.471,E2 -10552.471} C_VEL
LIN {X 0,Y 415.063,Z 529.365,A -85,B 0,C 180,E1 -10555.849,E2 -10555.849} C_VEL
LIN {X 0,Y 414.739,Z 524.932,A -85,B 0,C 180,E1 -10556.682,E2 -10556.682} C_VEL
LIN {X 0,Y 411.768,Z 510.803,A -85,B 0,C 180,E1 -10559.488,E2 -10559.488} C_VEL
LIN {X 0,Y 411.218,Z 508.263,A -85,B 0,C 180,E1 -10560.028,E2 -10560.028} C_VEL
LIN {X 0,Y 411.204,Z 508.267,A -85,B 0,C 180,E1 -10563.155,E2 -10563.155} C_VEL
LIN {X 0,Y 411.19,Z 508.259,A -85,B 0,C 180,E1 -10566.552,E2 -10566.552} C_VEL
LIN {X 0,Y 411.215,Z 508.254,A -85,B 0,C 180,E1 -10569.728,E2 -10569.728} C_VEL
LIN {X 0,Y 411.174,Z 508.265,A -85,B 0,C 180,E1 -10573.132,E2 -10573.132} C_VEL
LIN {X 0,Y 411.164,Z 508.268,A -85,B 0,C 180,E1 -10575.88,E2 -10575.88} C_VEL
LIN {X 0,Y 411.195,Z 508.257,A -85,B 0,C 180,E1 -10578.765,E2 -10578.765} C_VEL
LIN {X 0,Y 411.198,Z 508.259,A -85,B 0,C 180,E1 -10582.027,E2 -10582.027} C_VEL
LIN {X 0,Y 411.2,Z 508.263,A -85,B 0,C 180,E1 -10585.666,E2 -10585.666} C_VEL
LIN {X 0,Y 411.19,Z 508.255,A -85,B 0,C 180,E1 -10589.153,E2 -10589.153} C_VEL
LIN {X 0,Y 411.252,Z 508.255,A -85,B 0,C 180,E1 -10592.522,E2 -10592.522} C_VEL
LIN {X 0,Y 411.212,Z 508.245,A -85,B 0,C 180,E1 -10595.784,E2 -10595.784} C_VEL
LIN {X 0,Y 411.188,Z 508.264,A -85,B 0,C 180,E1 -10598.966,E2 -10598.966} C_VEL
LIN {X 0,Y 411.244,Z 508.247,A -85,B 0,C 180,E1 -10602.085,E2 -10602.085} C_VEL
LIN {X 0,Y 411.253,Z 508.249,A -85,B 0,C 180,E1 -10605.147,E2 -10605.147} C_VEL
LIN {X 0,Y 411.291,Z 508.249,A -85,B 0,C 180,E1 -10608.168,E2 -10608.168} C_VEL
LIN {X 0,Y 411.434,Z 508.216,A -85,B 0,C 180,E1 -10612.186,E2 -10612.186} C_VEL
LIN {X 0,Y 411.484,Z 508.222,A -85,B 0,C 180,E1 -10614.118,E2 -10614.118} C_VEL
LIN {X 0,Y 411.505,Z 508.217,A -85,B 0,C 180,E1 -10618.043,E2 -10618.043} C_VEL
LIN {X 0,Y 411.635,Z 508.187,A -85,B 0,C 180,E1 -10620,E2 -10620} C_VEL
LIN {X 0,Y 411.46,Z 508.229,A -85,B 0,C 180,E1 -10622.937,E2 -10622.937} C_VEL
LIN {X 0,Y 411.447,Z 508.224,A -85,B 0,C 180,E1 -10626.61,E2 -10626.61} C_VEL
LIN {X 0,Y 411.286,Z 508.244,A -85,B 0,C 180,E1 -10629.839,E2 -10629.839} C_VEL
LIN {X 0,Y 411.297,Z 508.253,A -85,B 0,C 180,E1 -10633.105,E2 -10633.105} C_VEL
LIN {X 0,Y 411.25,Z 508.243,A -85,B 0,C 180,E1 -10636.889,E2 -10636.889} C_VEL
LIN {X 0,Y 411.223,Z 508.258,A -85,B 0,C 180,E1 -10639.988,E2 -10639.988} C_VEL
LIN {X 0,Y 411.196,Z 508.253,A -85,B 0,C 180,E1 -10643.148,E2 -10643.148} C_VEL
LIN {X 0,Y 411.232,Z 508.258,A -85,B 0,C 180,E1 -10646.382,E2 -10646.382} C_VEL
LIN {X 0,Y 411.206,Z 508.253,A -85,B 0,C 180,E1 -10649.713,E2 -10649.713} C_VEL
LIN {X 0,Y 411.202,Z 508.263,A -85,B 0,C 180,E1 -10653.157,E2 -10653.157} C_VEL
LIN {X 0,Y 411.191,Z 508.264,A -85,B 0,C 180,E1 -10656.554,E2 -10656.554} C_VEL
LIN {X 0,Y 411.212,Z 508.259,A -85,B 0,C 180,E1 -10659.729,E2 -10659.729} C_VEL
LIN {X 0,Y 411.175,Z 508.266,A -85,B 0,C 180,E1 -10663.134,E2 -10663.134} C_VEL
LIN {X 0,Y 411.173,Z 508.266,A -85,B 0,C 180,E1 -10665.881,E2 -10665.881} C_VEL
LIN {X 0,Y 411.164,Z 508.271,A -85,B 0,C 180,E1 -10668.772,E2 -10668.772} C_VEL
LIN {X 0,Y 411.205,Z 508.259,A -85,B 0,C 180,E1 -10671.832,E2 -10671.832} C_VEL
LIN {X 0,Y 411.211,Z 508.256,A -85,B 0,C 180,E1 -10675.122,E2 -10675.122} C_VEL
LIN {X 0,Y 411.166,Z 508.261,A -85,B 0,C 180,E1 -10678.004,E2 -10678.004} C_VEL
LIN {X 0,Y 411.286,Z 508.41,A -85,B 0,C 180,E1 -10681.114,E2 -10681.114} C_VEL
LIN {X 0,Y 414.124,Z 521.751,A -85,B 0,C 180,E1 -10683.818,E2 -10683.818} C_VEL
LIN {X 0,Y 414.495,Z 526.263,A -85,B 0,C 180,E1 -10684.689,E2 -10684.689} C_VEL
LIN {X 0,Y 413.705,Z 545.019,A -85,B 0,C 180,E1 -10688.054,E2 -10688.054} C_VEL
LIN {X 0,Y 413.555,Z 547.999,A -85,B 0,C 180,E1 -10688.566,E2 -10688.566} C_VEL
LIN {X 0,Y 417.448,Z 569.02,A -85,B 0,C 180,E1 -10689.157,E2 -10689.157} C_VEL
LIN {X 0,Y 416.307,Z 657.665,A -85,B 0,C 180,E1 -10690.717,E2 -10690.717} C_VEL
LIN {X 0,Y 415.887,Z 671.094,A -85,B 0,C 180,E1 -10691.146,E2 -10691.146} C_VEL
LIN {X 0,Y 415.361,Z 684.18,A -85,B 0,C 180,E1 -10691.792,E2 -10691.792} C_VEL
LIN {X 0,Y 414.766,Z 694.889,A -85,B 0,C 180,E1 -10692.497,E2 -10692.497} C_VEL
LIN {X 0,Y 414.04,Z 705.254,A -85,B 0,C 180,E1 -10693.355,E2 -10693.355} C_VEL
LIN {X 0,Y 413.145,Z 715.902,A -85,B 0,C 180,E1 -10694.46,E2 -10694.46} C_VEL
LIN {X 0,Y 412.379,Z 725.444,A -85,B 0,C 180,E1 -10695.693,E2 -10695.693} C_VEL
LIN {X 0,Y 411.796,Z 733.371,A -85,B 0,C 180,E1 -10696.949,E2 -10696.949} C_VEL
LIN {X 0,Y 411.259,Z 740.935,A -85,B 0,C 180,E1 -10698.417,E2 -10698.417} C_VEL
LIN {X 0,Y 410.772,Z 746.131,A -85,B 0,C 180,E1 -10699.651,E2 -10699.651} C_VEL
LIN {X 0,Y 410.434,Z 751.182,A -85,B 0,C 180,E1 -10701.135,E2 -10701.135} C_VEL
LIN {X 0,Y 410.173,Z 755.675,A -85,B 0,C 180,E1 -10702.902,E2 -10702.902} C_VEL
LIN {X 0,Y 409.458,Z 757.266,A -85,B 0,C 180,E1 -10703.691,E2 -10703.691} C_VEL
LIN {X 0,Y 406.485,Z 759.363,A -85,B 0,C 180,E1 -10704.987,E2 -10704.987} C_VEL
LIN {X 0,Y 403.993,Z 760.49,A -85,B 0,C 180,E1 -10706.047,E2 -10706.047} C_VEL
LIN {X 0,Y 402.933,Z 760.96,A -85,B 0,C 180,E1 -10706.874,E2 -10706.874} C_VEL
LIN {X 0,Y 402.853,Z 761.035,A -85,B 0,C 180,E1 -10707.155,E2 -10707.155} C_VEL
LIN {X 0,Y 402.912,Z 761.193,A -85,B 0,C 180,E1 -10708.001,E2 -10708.001} C_VEL
LIN {X 0,Y 402.854,Z 760.341,A -85,B 0,C 180,E1 -10710,E2 -10710} C_VEL
LIN {X 0,Y 402.878,Z 759.344,A -85,B 0,C 180,E1 -10711,E2 -10711} C_VEL
LIN {X 0,Y 403.008,Z 757.919,A -85,B 0,C 180,E1 -10711.999,E2 -10711.999} C_VEL
LIN {X 0,Y 403.227,Z 754.989,A -85,B 0,C 180,E1 -10713.497,E2 -10713.497} C_VEL
LIN {X 0,Y 403.313,Z 751.029,A -85,B 0,C 180,E1 -10714.998,E2 -10714.998} C_VEL
LIN {X 0,Y 403.746,Z 745.91,A -85,B 0,C 180,E1 -10716.496,E2 -10716.496} C_VEL
LIN {X 0,Y 404.197,Z 739.484,A -85,B 0,C 180,E1 -10717.996,E2 -10717.996} C_VEL
LIN {X 0,Y 404.813,Z 731.5,A -85,B 0,C 180,E1 -10719.493,E2 -10719.493} C_VEL
LIN {X 0,Y 405.494,Z 723.324,A -85,B 0,C 180,E1 -10720.738,E2 -10720.738} C_VEL
LIN {X 0,Y 406.302,Z 713.255,A -85,B 0,C 180,E1 -10721.98,E2 -10721.98} C_VEL
LIN {X 0,Y 407.091,Z 701.985,A -85,B 0,C 180,E1 -10723.096,E2 -10723.096} C_VEL
LIN {X 0,Y 407.733,Z 690.822,A -85,B 0,C 180,E1 -10723.964,E2 -10723.964} C_VEL
LIN {X 0,Y 408.507,Z 678.225,A -85,B 0,C 180,E1 -10724.7,E2 -10724.7} C_VEL
LIN {X 0,Y 408.926,Z 665.729,A -85,B 0,C 180,E1 -10725.23,E2 -10725.23} C_VEL
LIN {X 0,Y 409.183,Z 653.2,A -85,B 0,C 180,E1 -10725.564,E2 -10725.564} C_VEL
LIN {X 0,Y 410.181,Z 569.757,A -85,B 0,C 180,E1 -10727.031,E2 -10727.031} C_VEL
LIN {X 0,Y 406.452,Z 548.128,A -85,B 0,C 180,E1 -10727.618,E2 -10727.618} C_VEL
LIN {X 0,Y 407.092,Z 530.812,A -85,B 0,C 180,E1 -10730.709,E2 -10730.709} C_VEL
LIN {X 0,Y 407.361,Z 524.996,A -85,B 0,C 180,E1 -10731.772,E2 -10731.772} C_VEL
LIN {X 0,Y 404.854,Z 512.021,A -85,B 0,C 180,E1 -10734.348,E2 -10734.348} C_VEL
LIN {X 0,Y 404.202,Z 509.144,A -85,B 0,C 180,E1 -10734.952,E2 -10734.952} C_VEL
LIN {X 0,Y 404.197,Z 509.137,A -85,B 0,C 180,E1 -10737.999,E2 -10737.999} C_VEL
LIN {X 0,Y 404.141,Z 509.146,A -85,B 0,C 180,E1 -10741.557,E2 -10741.557} C_VEL
LIN {X 0,Y 404.185,Z 509.141,A -85,B 0,C 180,E1 -10745.015,E2 -10745.015} C_VEL
LIN {X 0,Y 404.153,Z 509.145,A -85,B 0,C 180,E1 -10748.756,E2 -10748.756} C_VEL
LIN {X 0,Y 404.181,Z 509.136,A -85,B 0,C 180,E1 -10751.608,E2 -10751.608} C_VEL
LIN {X 0,Y 404.188,Z 509.132,A -85,B 0,C 180,E1 -10754.528,E2 -10754.528} C_VEL
LIN {X 0,Y 404.137,Z 509.143,A -85,B 0,C 180,E1 -10757.295,E2 -10757.295} C_VEL
LIN {X 0,Y 404.166,Z 509.138,A -85,B 0,C 180,E1 -10759.954,E2 -10759.954} C_VEL
LIN {X 0,Y 404.136,Z 509.146,A -85,B 0,C 180,E1 -10763.123,E2 -10763.123} C_VEL
LIN {X 0,Y 404.182,Z 509.141,A -85,B 0,C 180,E1 -10764.622,E2 -10764.622} C_VEL
LIN {X 0,Y 407.346,Z 518.251,A -85,B 0,C 180,E1 -10764.975,E2 -10764.975} C_VEL
LIN {X 0,Y 410.008,Z 526.347,A -85,B 0,C 180,E1 -10765.259,E2 -10765.259} C_VEL
LIN {X 0,Y 408.423,Z 614.572,A -85,B 0,C 180,E1 -10767.052,E2 -10767.052} C_VEL
LIN {X 0,Y 408.072,Z 628.566,A -85,B 0,C 180,E1 -10767.552,E2 -10767.552} C_VEL
LIN {X 0,Y 407.615,Z 640.954,A -85,B 0,C 180,E1 -10768.2,E2 -10768.2} C_VEL
LIN {X 0,Y 406.974,Z 653.603,A -85,B 0,C 180,E1 -10769.086,E2 -10769.086} C_VEL
LIN {X 0,Y 406.371,Z 664.309,A -85,B 0,C 180,E1 -10770.041,E2 -10770.041} C_VEL
LIN {X 0,Y 405.76,Z 674.165,A -85,B 0,C 180,E1 -10771.13,E2 -10771.13} C_VEL
LIN {X 0,Y 405.139,Z 683.514,A -85,B 0,C 180,E1 -10772.4,E2 -10772.4} C_VEL
LIN {X 0,Y 404.586,Z 691.422,A -85,B 0,C 180,E1 -10773.707,E2 -10773.707} C_VEL
LIN {X 0,Y 404.171,Z 697.912,A -85,B 0,C 180,E1 -10775.01,E2 -10775.01} C_VEL
LIN {X 0,Y 403.826,Z 703.599,A -85,B 0,C 180,E1 -10776.404,E2 -10776.404} C_VEL
LIN {X 0,Y 403.508,Z 708.797,A -85,B 0,C 180,E1 -10778.008,E2 -10778.008} C_VEL
LIN {X 0,Y 403.276,Z 712.661,A -85,B 0,C 180,E1 -10779.601,E2 -10779.601} C_VEL
LIN {X 0,Y 403.145,Z 714.549,A -85,B 0,C 180,E1 -10780.656,E2 -10780.656} C_VEL
LIN {X 0,Y 403.054,Z 715.983,A -85,B 0,C 180,E1 -10781.707,E2 -10781.707} C_VEL
LIN {X 0,Y 403.054,Z 717.368,A -85,B 0,C 180,E1 -10783.537,E2 -10783.537} C_VEL
LIN {X 0,Y 403.019,Z 717.492,A -85,B 0,C 180,E1 -10784.836,E2 -10784.836} C_VEL
LIN {X 0,Y 403.08,Z 717.115,A -85,B 0,C 180,E1 -10785.871,E2 -10785.871} C_VEL
LIN {X 0,Y 403.248,Z 715.699,A -85,B 0,C 180,E1 -10787.414,E2 -10787.414} C_VEL
LIN {X 0,Y 403.558,Z 712.21,A -85,B 0,C 180,E1 -10789.463,E2 -10789.463} C_VEL
LIN {X 0,Y 403.901,Z 708.362,A -85,B 0,C 180,E1 -10790.99,E2 -10790.99} C_VEL
LIN {X 0,Y 404.328,Z 703.252,A -85,B 0,C 180,E1 -10792.537,E2 -10792.537} C_VEL
LIN {X 0,Y 404.861,Z 697.012,A -85,B 0,C 180,E1 -10794.021,E2 -10794.021} C_VEL
LIN {X 0,Y 405.53,Z 689.085,A -85,B 0,C 180,E1 -10795.527,E2 -10795.527} C_VEL
LIN {X 0,Y 406.205,Z 681,A -85,B 0,C 180,E1 -10796.776,E2 -10796.776} C_VEL
LIN {X 0,Y 406.939,Z 671.164,A -85,B 0,C 180,E1 -10798.02,E2 -10798.02} C_VEL
LIN {X 0,Y 407.719,Z 661.392,A -85,B 0,C 180,E1 -10799.012,E2 -10799.012} C_VEL
LIN {X 0,Y 408.373,Z 650.889,A -85,B 0,C 180,E1 -10799.877,E2 -10799.877} C_VEL
LIN {X 0,Y 409.048,Z 638.399,A -85,B 0,C 180,E1 -10800.677,E2 -10800.677} C_VEL
LIN {X 0,Y 409.452,Z 626.078,A -85,B 0,C 180,E1 -10801.26,E2 -10801.26} C_VEL
LIN {X 0,Y 409.765,Z 613.383,A -85,B 0,C 180,E1 -10801.658,E2 -10801.658} C_VEL
LIN {X 0,Y 411.787,Z 528.526,A -85,B 0,C 180,E1 -10803.48,E2 -10803.48} C_VEL
LIN {X 0,Y 408.306,Z 519.541,A -85,B 0,C 180,E1 -10803.922,E2 -10803.922} C_VEL
LIN {X 0,Y 404.793,Z 511.757,A -85,B 0,C 180,E1 -10804.356,E2 -10804.356} C_VEL
LIN {X 0,Y 404.316,Z 509.126,A -85,B 0,C 180,E1 -10805.236,E2 -10805.236} C_VEL
LIN {X 0,Y 404.414,Z 509.111,A -85,B 0,C 180,E1 -10807.991,E2 -10807.991} C_VEL
LIN {X 0,Y 404.263,Z 509.128,A -85,B 0,C 180,E1 -10812.041,E2 -10812.041} C_VEL
LIN {X 0,Y 404.2,Z 509.137,A -85,B 0,C 180,E1 -10815.118,E2 -10815.118} C_VEL
LIN {X 0,Y 404.202,Z 509.133,A -85,B 0,C 180,E1 -10818.238,E2 -10818.238} C_VEL
LIN {X 0,Y 404.13,Z 509.144,A -85,B 0,C 180,E1 -10821.42,E2 -10821.42} C_VEL
LIN {X 0,Y 404.169,Z 509.139,A -85,B 0,C 180,E1 -10824.666,E2 -10824.666} C_VEL
LIN {X 0,Y 404.191,Z 509.132,A -85,B 0,C 180,E1 -10828,E2 -10828} C_VEL
LIN {X 0,Y 404.136,Z 509.139,A -85,B 0,C 180,E1 -10831.559,E2 -10831.559} C_VEL
LIN {X 0,Y 404.179,Z 509.14,A -85,B 0,C 180,E1 -10835.017,E2 -10835.017} C_VEL
LIN {X 0,Y 404.153,Z 509.141,A -85,B 0,C 180,E1 -10838.757,E2 -10838.757} C_VEL
LIN {X 0,Y 404.118,Z 509.145,A -85,B 0,C 180,E1 -10841.6,E2 -10841.6} C_VEL
LIN {X 0,Y 404.142,Z 509.143,A -85,B 0,C 180,E1 -10844.523,E2 -10844.523} C_VEL
LIN {X 0,Y 404.135,Z 509.146,A -85,B 0,C 180,E1 -10847.297,E2 -10847.297} C_VEL
LIN {X 0,Y 404.165,Z 509.141,A -85,B 0,C 180,E1 -10849.956,E2 -10849.956} C_VEL
LIN {X 0,Y 404.137,Z 509.146,A -85,B 0,C 180,E1 -10853.125,E2 -10853.125} C_VEL
LIN {X 0,Y 404.143,Z 509.146,A -85,B 0,C 180,E1 -10856.188,E2 -10856.188} C_VEL
LIN {X 0,Y 404.167,Z 509.265,A -85,B 0,C 180,E1 -10858.885,E2 -10858.885} C_VEL
LIN {X 0,Y 406.654,Z 519.387,A -85,B 0,C 180,E1 -10861.286,E2 -10861.286} C_VEL
LIN {X 0,Y 408.49,Z 529.168,A -85,B 0,C 180,E1 -10863.428,E2 -10863.428} C_VEL
LIN {X 0,Y 407.917,Z 537.448,A -85,B 0,C 180,E1 -10865.033,E2 -10865.033} C_VEL
LIN {X 0,Y 406.67,Z 552.764,A -85,B 0,C 180,E1 -10867.922,E2 -10867.922} C_VEL
LIN {X 0,Y 406.012,Z 562.632,A -85,B 0,C 180,E1 -10869.73,E2 -10869.73} C_VEL
LIN {X 0,Y 409.332,Z 584.332,A -85,B 0,C 180,E1 -10870.445,E2 -10870.445} C_VEL
LIN {X 0,Y 410.671,Z 598.193,A -85,B 0,C 180,E1 -10870.847,E2 -10870.847} C_VEL
LIN {X 0,Y 409.049,Z 674.52,A -85,B 0,C 180,E1 -10872.47,E2 -10872.47} C_VEL
LIN {X 0,Y 408.451,Z 687.432,A -85,B 0,C 180,E1 -10872.928,E2 -10872.928} C_VEL
LIN {X 0,Y 407.425,Z 706.07,A -85,B 0,C 180,E1 -10873.85,E2 -10873.85} C_VEL
LIN {X 0,Y 406.687,Z 717.341,A -85,B 0,C 180,E1 -10874.592,E2 -10874.592} C_VEL
LIN {X 0,Y 405.989,Z 728.158,A -85,B 0,C 180,E1 -10875.514,E2 -10875.514} C_VEL
LIN {X 0,Y 405.365,Z 737.581,A -85,B 0,C 180,E1 -10876.51,E2 -10876.51} C_VEL
LIN {X 0,Y 404.667,Z 746.938,A -85,B 0,C 180,E1 -10877.717,E2 -10877.717} C_VEL
LIN {X 0,Y 404.058,Z 754.907,A -85,B 0,C 180,E1 -10878.97,E2 -10878.97} C_VEL
LIN {X 0,Y 403.569,Z 762.669,A -85,B 0,C 180,E1 -10880.478,E2 -10880.478} C_VEL
LIN {X 0,Y 403.232,Z 768.861,A -85,B 0,C 180,E1 -10881.985,E2 -10881.985} C_VEL
LIN {X 0,Y 403.006,Z 774.443,A -85,B 0,C 180,E1 -10883.732,E2 -10883.732} C_VEL
LIN {X 0,Y 402.983,Z 777.515,A -85,B 0,C 180,E1 -10884.998,E2 -10884.998} C_VEL
LIN {X 0,Y 402.88,Z 779.442,A -85,B 0,C 180,E1 -10885.999,E2 -10885.999} C_VEL
LIN {X 0,Y 402.895,Z 780.934,A -85,B 0,C 180,E1 -10887,E2 -10887} C_VEL
LIN {X 0,Y 402.94,Z 781.974,A -85,B 0,C 180,E1 -10888.001,E2 -10888.001} C_VEL
LIN {X 0,Y 402.861,Z 782.871,A -85,B 0,C 180,E1 -10890,E2 -10890} C_VEL
LIN {X 0,Y 402.873,Z 782.7,A -85,B 0,C 180,E1 -10891,E2 -10891} C_VEL
LIN {X 0,Y 402.94,Z 782.111,A -85,B 0,C 180,E1 -10891.999,E2 -10891.999} C_VEL
LIN {X 0,Y 402.897,Z 781.128,A -85,B 0,C 180,E1 -10893,E2 -10893} C_VEL
LIN {X 0,Y 402.882,Z 779.744,A -85,B 0,C 180,E1 -10894.001,E2 -10894.001} C_VEL
LIN {X 0,Y 402.969,Z 776.821,A -85,B 0,C 180,E1 -10895.504,E2 -10895.504} C_VEL
LIN {X 0,Y 403.098,Z 772.848,A -85,B 0,C 180,E1 -10897.01,E2 -10897.01} C_VEL
LIN {X 0,Y 403.404,Z 766.693,A -85,B 0,C 180,E1 -10898.768,E2 -10898.768} C_VEL
LIN {X 0,Y 403.869,Z 759.968,A -85,B 0,C 180,E1 -10900.274,E2 -10900.274} C_VEL
LIN {X 0,Y 404.491,Z 751.6,A -85,B 0,C 180,E1 -10901.78,E2 -10901.78} C_VEL
LIN {X 0,Y 405.18,Z 742.949,A -85,B 0,C 180,E1 -10903.031,E2 -10903.031} C_VEL
LIN {X 0,Y 405.974,Z 732.52,A -85,B 0,C 180,E1 -10904.255,E2 -10904.255} C_VEL
LIN {X 0,Y 406.776,Z 721.627,A -85,B 0,C 180,E1 -10905.276,E2 -10905.276} C_VEL
LIN {X 0,Y 407.572,Z 709.639,A -85,B 0,C 180,E1 -10906.144,E2 -10906.144} C_VEL
LIN {X 0,Y 408.287,Z 697.115,A -85,B 0,C 180,E1 -10906.822,E2 -10906.822} C_VEL
LIN {X 0,Y 408.817,Z 684.781,A -85,B 0,C 180,E1 -10907.282,E2 -10907.282} C_VEL
LIN {X 0,Y 409.149,Z 670.896,A -85,B 0,C 180,E1 -10907.59,E2 -10907.59} C_VEL
LIN {X 0,Y 409.823,Z 595.789,A -85,B 0,C 180,E1 -10908.918,E2 -10908.918} C_VEL
LIN {X 0,Y 405.728,Z 565.172,A -85,B 0,C 180,E1 -10909.703,E2 -10909.703} C_VEL
LIN {X 0,Y 406.98,Z 546.109,A -85,B 0,C 180,E1 -10913.132,E2 -10913.132} C_VEL
LIN {X 0,Y 408.18,Z 528.863,A -85,B 0,C 180,E1 -10916.279,E2 -10916.279} C_VEL
LIN {X 0,Y 406.031,Z 517.695,A -85,B 0,C 180,E1 -10918.496,E2 -10918.496} C_VEL
LIN {X 0,Y 404.173,Z 509.141,A -85,B 0,C 180,E1 -10920.282,E2 -10920.282} C_VEL
LIN {X 0,Y 404.143,Z 509.143,A -85,B 0,C 180,E1 -10923.812,E2 -10923.812} C_VEL
LIN {X 0,Y 404.133,Z 509.13,A -85,B 0,C 180,E1 -10926.874,E2 -10926.874} C_VEL
LIN {X 0,Y 404.145,Z 509.137,A -85,B 0,C 180,E1 -10930.08,E2 -10930.08} C_VEL
LIN {X 0,Y 404.153,Z 509.14,A -85,B 0,C 180,E1 -10933.084,E2 -10933.084} C_VEL
LIN {X 0,Y 404.144,Z 509.142,A -85,B 0,C 180,E1 -10935.925,E2 -10935.925} C_VEL
LIN {X 0,Y 404.146,Z 509.134,A -85,B 0,C 180,E1 -10938.638,E2 -10938.638} C_VEL
LIN {X 0,Y 404.156,Z 509.14,A -85,B 0,C 180,E1 -10941.49,E2 -10941.49} C_VEL
LIN {X 0,Y 404.179,Z 509.135,A -85,B 0,C 180,E1 -10944.983,E2 -10944.983} C_VEL
LIN {X 0,Y 404.139,Z 509.137,A -85,B 0,C 180,E1 -10948.554,E2 -10948.554} C_VEL
LIN {X 0,Y 404.191,Z 509.134,A -85,B 0,C 180,E1 -10952,E2 -10952} C_VEL
LIN {X 0,Y 404.166,Z 509.125,A -85,B 0,C 180,E1 -10955.334,E2 -10955.334} C_VEL
LIN {X 0,Y 404.13,Z 509.14,A -85,B 0,C 180,E1 -10958.58,E2 -10958.58} C_VEL
LIN {X 0,Y 404.202,Z 509.125,A -85,B 0,C 180,E1 -10961.762,E2 -10961.762} C_VEL
LIN {X 0,Y 404.198,Z 509.124,A -85,B 0,C 180,E1 -10964.882,E2 -10964.882} C_VEL
LIN {X 0,Y 404.262,Z 509.125,A -85,B 0,C 180,E1 -10967.959,E2 -10967.959} C_VEL
LIN {X 0,Y 404.375,Z 509.095,A -85,B 0,C 180,E1 -10972.008,E2 -10972.008} C_VEL
LIN {X 0,Y 404.43,Z 509.101,A -85,B 0,C 180,E1 -10974.015,E2 -10974.015} C_VEL
LIN {X 0,Y 404.474,Z 509.093,A -85,B 0,C 180,E1 -10978.009,E2 -10978.009} C_VEL
LIN {X 0,Y 404.604,Z 509.062,A -85,B 0,C 180,E1 -10980,E2 -10980} C_VEL
LIN {X 0,Y 404.417,Z 509.106,A -85,B 0,C 180,E1 -10982.989,E2 -10982.989} C_VEL
LIN {X 0,Y 404.393,Z 509.101,A -85,B 0,C 180,E1 -10986.607,E2 -10986.607} C_VEL
LIN {X 0,Y 404.283,Z 509.109,A -85,B 0,C 180,E1 -10989.001,E2 -10989.001} C_VEL
LIN {X 0,Y 404.249,Z 509.127,A -85,B 0,C 180,E1 -10992.042,E2 -10992.042} C_VEL
LIN {X 0,Y 404.198,Z 509.124,A -85,B 0,C 180,E1 -10995.119,E2 -10995.119} C_VEL
LIN {X 0,Y 404.203,Z 509.129,A -85,B 0,C 180,E1 -10998.239,E2 -10998.239} C_VEL
LIN {X 0,Y 404.131,Z 509.139,A -85,B 0,C 180,E1 -11001.42,E2 -11001.42} C_VEL
LIN {X 0,Y 404.17,Z 509.131,A -85,B 0,C 180,E1 -11004.666,E2 -11004.666} C_VEL
LIN {X 0,Y 404.192,Z 509.131,A -85,B 0,C 180,E1 -11008,E2 -11008} C_VEL
LIN {X 0,Y 404.143,Z 509.142,A -85,B 0,C 180,E1 -11011.561,E2 -11011.561} C_VEL
LIN {X 0,Y 404.181,Z 509.133,A -85,B 0,C 180,E1 -11015.017,E2 -11015.017} C_VEL
LIN {X 0,Y 404.154,Z 509.143,A -85,B 0,C 180,E1 -11018.758,E2 -11018.758} C_VEL
LIN {X 0,Y 404.121,Z 509.148,A -85,B 0,C 180,E1 -11021.601,E2 -11021.601} C_VEL
LIN {X 0,Y 404.148,Z 509.141,A -85,B 0,C 180,E1 -11024.524,E2 -11024.524} C_VEL
LIN {X 0,Y 404.138,Z 509.144,A -85,B 0,C 180,E1 -11027.297,E2 -11027.297} C_VEL
LIN {X 0,Y 404.168,Z 509.137,A -85,B 0,C 180,E1 -11029.956,E2 -11029.956} C_VEL
LIN {X 0,Y 404.136,Z 509.147,A -85,B 0,C 180,E1 -11033.126,E2 -11033.126} C_VEL
LIN {X 0,Y 404.145,Z 509.141,A -85,B 0,C 180,E1 -11036.189,E2 -11036.189} C_VEL
LIN {X 0,Y 404.147,Z 509.143,A -85,B 0,C 180,E1 -11039.716,E2 -11039.716} C_VEL
LIN {X 0,Y 404.218,Z 509.252,A -85,B 0,C 180,E1 -11040.805,E2 -11040.805} C_VEL
LIN {X 0,Y 406.892,Z 521.486,A -85,B 0,C 180,E1 -11043.316,E2 -11043.316} C_VEL
LIN {X 0,Y 407.614,Z 526.025,A -85,B 0,C 180,E1 -11044.226,E2 -11044.226} C_VEL
LIN {X 0,Y 407.1,Z 539.003,A -85,B 0,C 180,E1 -11046.606,E2 -11046.606} C_VEL
LIN {X 0,Y 406.7,Z 548.196,A -85,B 0,C 180,E1 -11048.222,E2 -11048.222} C_VEL
LIN {X 0,Y 410.764,Z 569.825,A -85,B 0,C 180,E1 -11048.837,E2 -11048.837} C_VEL
LIN {X 0,Y 409.558,Z 658.182,A -85,B 0,C 180,E1 -11050.419,E2 -11050.419} C_VEL
LIN {X 0,Y 409.139,Z 671.004,A -85,B 0,C 180,E1 -11050.835,E2 -11050.835} C_VEL
LIN {X 0,Y 408.684,Z 682.653,A -85,B 0,C 180,E1 -11051.404,E2 -11051.404} C_VEL
LIN {X 0,Y 407.982,Z 694.771,A -85,B 0,C 180,E1 -11052.196,E2 -11052.196} C_VEL
LIN {X 0,Y 407.225,Z 705.196,A -85,B 0,C 180,E1 -11053.069,E2 -11053.069} C_VEL
LIN {X 0,Y 406.268,Z 715.905,A -85,B 0,C 180,E1 -11054.19,E2 -11054.19} C_VEL
LIN {X 0,Y 405.48,Z 725.479,A -85,B 0,C 180,E1 -11055.445,E2 -11055.445} C_VEL
LIN {X 0,Y 404.812,Z 733.697,A -85,B 0,C 180,E1 -11056.766,E2 -11056.766} C_VEL
LIN {X 0,Y 404.277,Z 741.026,A -85,B 0,C 180,E1 -11058.214,E2 -11058.214} C_VEL
LIN {X 0,Y 403.753,Z 746.235,A -85,B 0,C 180,E1 -11059.469,E2 -11059.469} C_VEL
LIN {X 0,Y 403.396,Z 751.307,A -85,B 0,C 180,E1 -11060.979,E2 -11060.979} C_VEL
LIN {X 0,Y 403.091,Z 756.02,A -85,B 0,C 180,E1 -11062.873,E2 -11062.873} C_VEL
LIN {X 0,Y 402.989,Z 758.091,A -85,B 0,C 180,E1 -11063.994,E2 -11063.994} C_VEL
LIN {X 0,Y 402.945,Z 759.456,A -85,B 0,C 180,E1 -11064.997,E2 -11064.997} C_VEL
LIN {X 0,Y 402.852,Z 761.006,A -85,B 0,C 180,E1 -11067,E2 -11067} C_VEL
LIN {X 0,Y 402.853,Z 761.035,A -85,B 0,C 180,E1 -11067.155,E2 -11067.155} C_VEL
LIN {X 0,Y 402.188,Z 761.213,A -85,B 0,C 180,E1 -11067.991,E2 -11067.991} C_VEL
LIN {X 0,Y 399.297,Z 760.891,A -85,B 0,C 180,E1 -11069.348,E2 -11069.348} C_VEL
LIN {X 0,Y 396.888,Z 760.148,A -85,B 0,C 180,E1 -11070.439,E2 -11070.439} C_VEL
LIN {X 0,Y 395.911,Z 759.234,A -85,B 0,C 180,E1 -11071.277,E2 -11071.277} C_VEL
LIN {X 0,Y 395.864,Z 758.807,A -85,B 0,C 180,E1 -11071.558,E2 -11071.558} C_VEL
LIN {X 0,Y 396.164,Z 755.231,A -85,B 0,C 180,E1 -11073.56,E2 -11073.56} C_VEL
LIN {X 0,Y 396.253,Z 751.286,A -85,B 0,C 180,E1 -11075.088,E2 -11075.088} C_VEL
LIN {X 0,Y 396.697,Z 746.183,A -85,B 0,C 180,E1 -11076.612,E2 -11076.612} C_VEL
LIN {X 0,Y 397.285,Z 738.576,A -85,B 0,C 180,E1 -11078.392,E2 -11078.392} C_VEL
LIN {X 0,Y 397.811,Z 731.809,A -85,B 0,C 180,E1 -11079.662,E2 -11079.662} C_VEL
LIN {X 0,Y 398.545,Z 723.658,A -85,B 0,C 180,E1 -11080.927,E2 -11080.927} C_VEL
LIN {X 0,Y 399.365,Z 713.627,A -85,B 0,C 180,E1 -11082.191,E2 -11082.191} C_VEL
LIN {X 0,Y 400.203,Z 702.392,A -85,B 0,C 180,E1 -11083.326,E2 -11083.326} C_VEL
LIN {X 0,Y 400.884,Z 691.307,A -85,B 0,C 180,E1 -11084.207,E2 -11084.207} C_VEL
LIN {X 0,Y 401.685,Z 678.789,A -85,B 0,C 180,E1 -11084.955,E2 -11084.955} C_VEL
LIN {X 0,Y 402.116,Z 665.893,A -85,B 0,C 180,E1 -11085.515,E2 -11085.515} C_VEL
LIN {X 0,Y 402.433,Z 652.342,A -85,B 0,C 180,E1 -11085.873,E2 -11085.873} C_VEL
LIN {X 0,Y 403.452,Z 570.698,A -85,B 0,C 180,E1 -11087.329,E2 -11087.329} C_VEL
LIN {X 0,Y 399.588,Z 548.277,A -85,B 0,C 180,E1 -11087.951,E2 -11087.951} C_VEL
LIN {X 0,Y 400.332,Z 529.549,A -85,B 0,C 180,E1 -11091.324,E2 -11091.324} C_VEL
LIN {X 0,Y 400.477,Z 526.492,A -85,B 0,C 180,E1 -11091.895,E2 -11091.895} C_VEL
LIN {X 0,Y 397.903,Z 513.367,A -85,B 0,C 180,E1 -11094.523,E2 -11094.523} C_VEL
LIN {X 0,Y 397.18,Z 510.017,A -85,B 0,C 180,E1 -11095.234,E2 -11095.234} C_VEL
LIN {X 0,Y 397.164,Z 510.014,A -85,B 0,C 180,E1 -11097.775,E2 -11097.775} C_VEL
LIN {X 0,Y 397.08,Z 510.025,A -85,B 0,C 180,E1 -11100.881,E2 -11100.881} C_VEL
LIN {X 0,Y 397.126,Z 510.015,A -85,B 0,C 180,E1 -11104.492,E2 -11104.492} C_VEL
LIN {X 0,Y 397.102,Z 510.019,A -85,B 0,C 180,E1 -11108.274,E2 -11108.274} C_VEL
LIN {X 0,Y 397.148,Z 510.012,A -85,B 0,C 180,E1 -11111.991,E2 -11111.991} C_VEL
LIN {X 0,Y 397.111,Z 510.01,A -85,B 0,C 180,E1 -11115.064,E2 -11115.064} C_VEL
LIN {X 0,Y 397.065,Z 510.023,A -85,B 0,C 180,E1 -11118.02,E2 -11118.02} C_VEL
LIN {X 0,Y 397.129,Z 510.018,A -85,B 0,C 180,E1 -11121.137,E2 -11121.137} C_VEL
LIN {X 0,Y 397.123,Z 510.02,A -85,B 0,C 180,E1 -11124.335,E2 -11124.335} C_VEL
LIN {X 0,Y 401.816,Z 523.248,A -85,B 0,C 180,E1 -11124.852,E2 -11124.852} C_VEL
LIN {X 0,Y 403.175,Z 527.967,A -85,B 0,C 180,E1 -11125.011,E2 -11125.011} C_VEL
LIN {X 0,Y 401.506,Z 615.604,A -85,B 0,C 180,E1 -11126.838,E2 -11126.838} C_VEL
LIN {X 0,Y 401.18,Z 629.047,A -85,B 0,C 180,E1 -11127.332,E2 -11127.332} C_VEL
LIN {X 0,Y 400.692,Z 642.033,A -85,B 0,C 180,E1 -11128.029,E2 -11128.029} C_VEL
LIN {X 0,Y 400.009,Z 654.552,A -85,B 0,C 180,E1 -11128.928,E2 -11128.928} C_VEL
LIN {X 0,Y 399.382,Z 665.253,A -85,B 0,C 180,E1 -11129.907,E2 -11129.907} C_VEL
LIN {X 0,Y 398.715,Z 676.055,A -85,B 0,C 180,E1 -11131.149,E2 -11131.149} C_VEL
LIN {X 0,Y 398.054,Z 685.205,A -85,B 0,C 180,E1 -11132.441,E2 -11132.441} C_VEL
LIN {X 0,Y 397.507,Z 692.915,A -85,B 0,C 180,E1 -11133.768,E2 -11133.768} C_VEL
LIN {X 0,Y 397.007,Z 700.592,A -85,B 0,C 180,E1 -11135.417,E2 -11135.417} C_VEL
LIN {X 0,Y 396.626,Z 706.849,A -85,B 0,C 180,E1 -11137.13,E2 -11137.13} C_VEL
LIN {X 0,Y 396.338,Z 711.205,A -85,B 0,C 180,E1 -11138.684,E2 -11138.684} C_VEL
LIN {X 0,Y 396.121,Z 714.546,A -85,B 0,C 180,E1 -11140.299,E2 -11140.299} C_VEL
LIN {X 0,Y 395.992,Z 716.114,A -85,B 0,C 180,E1 -11141.369,E2 -11141.369} C_VEL
LIN {X 0,Y 395.98,Z 717.229,A -85,B 0,C 180,E1 -11142.439,E2 -11142.439} C_VEL
LIN {X 0,Y 395.982,Z 717.903,A -85,B 0,C 180,E1 -11143.502,E2 -11143.502} C_VEL
LIN {X 0,Y 395.967,Z 718.082,A -85,B 0,C 180,E1 -11144.559,E2 -11144.559} C_VEL
LIN {X 0,Y 395.98,Z 717.838,A -85,B 0,C 180,E1 -11145.612,E2 -11145.612} C_VEL
LIN {X 0,Y 396.169,Z 716.476,A -85,B 0,C 180,E1 -11147.335,E2 -11147.335} C_VEL
LIN {X 0,Y 396.474,Z 713.465,A -85,B 0,C 180,E1 -11149.273,E2 -11149.273} C_VEL
LIN {X 0,Y 396.814,Z 709.86,A -85,B 0,C 180,E1 -11150.828,E2 -11150.828} C_VEL
LIN {X 0,Y 397.283,Z 704.709,A -85,B 0,C 180,E1 -11152.49,E2 -11152.49} C_VEL
LIN {X 0,Y 397.919,Z 697.96,A -85,B 0,C 180,E1 -11154.171,E2 -11154.171} C_VEL
LIN {X 0,Y 398.626,Z 690.102,A -85,B 0,C 180,E1 -11155.703,E2 -11155.703} C_VEL
LIN {X 0,Y 399.335,Z 682.086,A -85,B 0,C 180,E1 -11156.973,E2 -11156.973} C_VEL
LIN {X 0,Y 400.112,Z 672.338,A -85,B 0,C 180,E1 -11158.239,E2 -11158.239} C_VEL
LIN {X 0,Y 400.976,Z 662.032,A -85,B 0,C 180,E1 -11159.309,E2 -11159.309} C_VEL
LIN {X 0,Y 401.721,Z 650.714,A -85,B 0,C 180,E1 -11160.25,E2 -11160.25} C_VEL
LIN {X 0,Y 402.392,Z 638.116,A -85,B 0,C 180,E1 -11161.063,E2 -11161.063} C_VEL
LIN {X 0,Y 402.891,Z 624.531,A -85,B 0,C 180,E1 -11161.687,E2 -11161.687} C_VEL
LIN {X 0,Y 403.19,Z 610.883,A -85,B 0,C 180,E1 -11162.091,E2 -11162.091} C_VEL
LIN {X 0,Y 405.275,Z 529.935,A -85,B 0,C 180,E1 -11163.867,E2 -11163.867} C_VEL
LIN {X 0,Y 401.507,Z 520.896,A -85,B 0,C 180,E1 -11164.352,E2 -11164.352} C_VEL
LIN {X 0,Y 397.773,Z 512.506,A -85,B 0,C 180,E1 -11164.846,E2 -11164.846} C_VEL
LIN {X 0,Y 397.363,Z 509.991,A -85,B 0,C 180,E1 -11165.709,E2 -11165.709} C_VEL
LIN {X 0,Y 397.369,Z 509.989,A -85,B 0,C 180,E1 -11168.134,E2 -11168.134} C_VEL
LIN {X 0,Y 397.222,Z 510.005,A -85,B 0,C 180,E1 -11172.258,E2 -11172.258} C_VEL
LIN {X 0,Y 397.172,Z 510.014,A -85,B 0,C 180,E1 -11175.392,E2 -11175.392} C_VEL
LIN {X 0,Y 397.154,Z 510.012,A -85,B 0,C 180,E1 -11178.574,E2 -11178.574} C_VEL
LIN {X 0,Y 397.089,Z 510.021,A -85,B 0,C 180,E1 -11181.819,E2 -11181.819} C_VEL
LIN {X 0,Y 397.149,Z 510.014,A -85,B 0,C 180,E1 -11185.132,E2 -11185.132} C_VEL
LIN {X 0,Y 397.156,Z 510.008,A -85,B 0,C 180,E1 -11187.777,E2 -11187.777} C_VEL
LIN {X 0,Y 397.078,Z 510.022,A -85,B 0,C 180,E1 -11190.882,E2 -11190.882} C_VEL
LIN {X 0,Y 397.119,Z 510.014,A -85,B 0,C 180,E1 -11194.494,E2 -11194.494} C_VEL
LIN {X 0,Y 397.101,Z 510.017,A -85,B 0,C 180,E1 -11198.275,E2 -11198.275} C_VEL
LIN {X 0,Y 397.083,Z 510.024,A -85,B 0,C 180,E1 -11200.909,E2 -11200.909} C_VEL
